KUKA KRL program: f1_Kuka_APT224T02S24.SRC

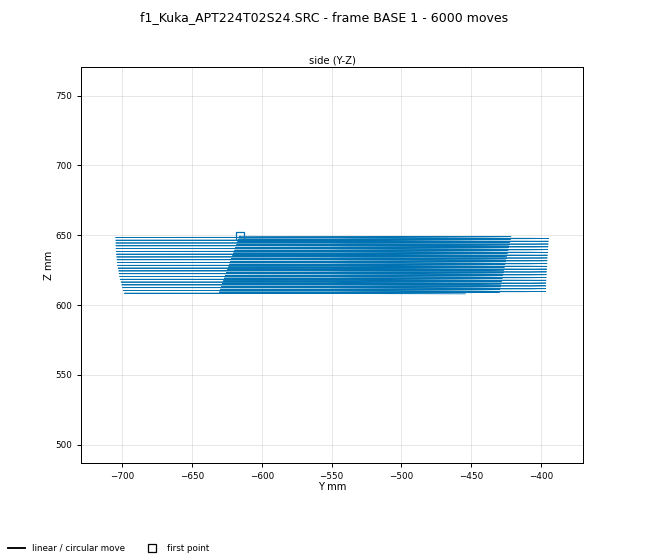
[picture p0: tool path of f1_Kuka_APT224T02S24.SRC in frame BASE 1, 6000 of 6001 moves have a stored position in this frame; points joined in program order, loops and branches not executed]
&ACCESS RVP
&REL 2
&PARAM TEMPLATE = C:\KRC\Roboter\Template\vorgabe
&PARAM EDITMASK = *
DEF f1_Kuka_APT224T02S24()


;FOLD INI;%{PE}%V3.2.0,%MKUKATPBASIS,%CINIT,%VCOMMON,%P
  ;FOLD BAS INI;%{E}%V3.2.0,%MKUKATPBASIS,%CINIT,%VINIT,%P
    GLOBAL INTERRUPT DECL 3 WHEN $STOPMESS==TRUE DO IR_STOPM ( )
    INTERRUPT ON 3
    BAS (#INITMOV,0 )
  ;ENDFOLD (BAS INI)
  ;FOLD USER INI;%{E}%V3.2.0,%MKUKATPUSER,%CINIT,%VINIT,%P
    ;Make your modifications here
  ;ENDFOLD (USER INI)
;ENDFOLD (INI)


;*** Make Null PTP Move
  PTP $pos_act

;*** Auto Load The Correct TOOL Data
  $tool=tool_data[2]

;*** Auto Load The Correct BASE Data
  $base=base_data[1]

  $ADVANCE = 5

;*** Restate Last Velocity
MMPM(30000.0)
SetRPM(8000)
LIN {X -0.107,Y -615.683,Z 649.293,A 0.000,B 0.000,C 90.000,E1 88.740} C_DIS
LIN {X -0.106,Y -616.052,Z 649.287,A 0.000,B 0.000,C 90.000,E1 87.707} C_DIS
LIN {X -0.093,Y -616.149,Z 649.281,A 0.000,B 0.000,C 90.000,E1 86.674} C_DIS
LIN {X 0.216,Y -615.988,Z 649.274,A 0.000,B 0.000,C 90.000,E1 85.355} C_DIS
LIN {X -0.079,Y -615.700,Z 649.270,A 0.000,B 0.000,C 90.000,E1 84.609} C_DIS
LIN {X -0.285,Y -615.137,Z 649.263,A 0.000,B 0.000,C 90.000,E1 83.337} C_DIS
LIN {X 0.118,Y -614.273,Z 649.256,A 0.000,B 0.000,C 90.000,E1 82.008} C_DIS
LIN {X 0.144,Y -613.216,Z 649.250,A 0.000,B 0.000,C 90.000,E1 80.971} C_DIS
LIN {X -0.008,Y -611.675,Z 649.243,A 0.000,B 0.000,C 90.000,E1 79.690} C_DIS
LIN {X -0.187,Y -609.834,Z 649.236,A 0.000,B 0.000,C 90.000,E1 78.409} C_DIS
LIN {X -0.275,Y -607.853,Z 649.228,A 0.000,B 0.000,C 90.000,E1 77.117} C_DIS
LIN {X 0.076,Y -605.171,Z 649.220,A 0.000,B 0.000,C 90.000,E1 75.519} C_DIS
LIN {X 0.063,Y -602.718,Z 649.212,A 0.000,B 0.000,C 90.000,E1 74.212} C_DIS
LIN {X 0.000,Y -600.058,Z 649.205,A 0.000,B 0.000,C 90.000,E1 72.906} C_DIS
LIN {X 0.062,Y -597.213,Z 649.198,A 0.000,B 0.000,C 90.000,E1 71.583} C_DIS
LIN {X 0.116,Y -595.336,Z 649.193,A 0.000,B 0.000,C 90.000,E1 70.786} C_DIS
LIN {X -0.045,Y -593.298,Z 649.189,A 0.000,B 0.000,C 90.000,E1 70.007} C_DIS
LIN {X -0.139,Y -590.246,Z 649.183,A 0.000,B 0.000,C 90.000,E1 68.954} C_DIS
LIN {X -0.032,Y -588.640,Z 649.180,A 0.000,B 0.000,C 90.000,E1 68.411} C_DIS
LIN {X -0.186,Y -584.996,Z 649.174,A 0.000,B 0.000,C 90.000,E1 67.358} C_DIS
LIN {X -0.157,Y -580.935,Z 649.168,A 0.000,B 0.000,C 90.000,E1 66.282} C_DIS
LIN {X -0.274,Y -577.678,Z 649.164,A 0.000,B 0.000,C 90.000,E1 65.485} C_DIS
LIN {X -0.191,Y -574.318,Z 649.159,A 0.000,B 0.000,C 90.000,E1 64.665} C_DIS
LIN {X 0.103,Y -570.576,Z 649.155,A 0.000,B 0.000,C 90.000,E1 63.819} C_DIS
LIN {X 0.189,Y -567.295,Z 649.151,A 0.000,B 0.000,C 90.000,E1 63.127} C_DIS
LIN {X -0.261,Y -563.689,Z 649.147,A 0.000,B 0.000,C 90.000,E1 62.487} C_DIS
LIN {X 0.018,Y -559.681,Z 649.143,A 0.000,B 0.000,C 90.000,E1 61.769} C_DIS
LIN {X 0.259,Y -555.194,Z 649.139,A 0.000,B 0.000,C 90.000,E1 61.051} C_DIS
LIN {X -0.181,Y -551.142,Z 649.136,A 0.000,B 0.000,C 90.000,E1 60.539} C_DIS
LIN {X 0.098,Y -546.732,Z 649.133,A 0.000,B 0.000,C 90.000,E1 59.950} C_DIS
LIN {X -0.119,Y -541.775,Z 649.130,A 0.000,B 0.000,C 90.000,E1 59.410} C_DIS
LIN {X -0.156,Y -537.571,Z 649.128,A 0.000,B 0.000,C 90.000,E1 58.997} C_DIS
LIN {X 0.112,Y -531.705,Z 649.125,A 0.000,B 0.000,C 90.000,E1 58.456} C_DIS
LIN {X 0.085,Y -525.967,Z 649.122,A 0.000,B 0.000,C 90.000,E1 57.995} C_DIS
LIN {X 0.245,Y -521.337,Z 649.121,A 0.000,B 0.000,C 90.000,E1 57.661} C_DIS
LIN {X -0.035,Y -515.202,Z 649.118,A 0.000,B 0.000,C 90.000,E1 57.296} C_DIS
LIN {X -0.193,Y -508.231,Z 649.116,A 0.000,B 0.000,C 90.000,E1 56.914} C_DIS
LIN {X 0.225,Y -501.476,Z 649.114,A 0.000,B 0.000,C 90.000,E1 56.501} C_DIS
LIN {X -0.128,Y -484.846,Z 649.109,A 0.000,B 0.000,C 90.000,E1 55.674} C_DIS
LIN {X -0.111,Y -464.619,Z 649.103,A 0.000,B 0.000,C 90.000,E1 54.609} C_DIS
LIN {X 0.001,Y -443.164,Z 649.097,A 0.000,B 0.000,C 90.000,E1 53.417} C_DIS
LIN {X -0.090,Y -435.744,Z 649.094,A 0.000,B 0.000,C 90.000,E1 53.004} C_DIS
LIN {X 0.128,Y -435.681,Z 649.094,A 0.000,B 0.000,C 90.000,E1 52.970} C_DIS
LIN {X -0.013,Y -431.775,Z 649.083,A 0.000,B 0.000,C 90.000,E1 50.964} C_DIS
LIN {X 0.166,Y -430.198,Z 649.079,A 0.000,B 0.000,C 90.000,E1 50.275} C_DIS
LIN {X -0.142,Y -421.586,Z 649.058,A 0.000,B 0.000,C 90.000,E1 46.458} C_DIS
LIN {X -0.193,Y -421.525,Z 649.057,A 0.000,B 0.000,C 90.000,E1 46.296} C_DIS
LIN {X -0.119,Y -421.750,Z 649.048,A 0.000,B 0.000,C 90.000,E1 44.595} C_DIS
LIN {X -0.046,Y -421.951,Z 649.038,A 0.000,B 0.000,C 90.000,E1 42.894} C_DIS
LIN {X 0.082,Y -422.604,Z 649.023,A 0.000,B 0.000,C 90.000,E1 40.172} C_DIS
LIN {X -0.082,Y -423.806,Z 649.006,A 0.000,B 0.000,C 90.000,E1 37.156} C_DIS
LIN {X 0.166,Y -424.678,Z 648.997,A 0.000,B 0.000,C 90.000,E1 35.438} C_DIS
LIN {X -0.039,Y -425.347,Z 648.990,A 0.000,B 0.000,C 90.000,E1 34.119} C_DIS
LIN {X 0.106,Y -426.158,Z 648.980,A 0.000,B 0.000,C 90.000,E1 32.418} C_DIS
LIN {X 0.029,Y -427.258,Z 648.967,A 0.000,B 0.000,C 90.000,E1 30.079} C_DIS
LIN {X -0.008,Y -427.926,Z 648.960,A 0.000,B 0.000,C 90.000,E1 28.743} C_DIS
LIN {X -0.083,Y -428.992,Z 648.949,A 0.000,B 0.000,C 90.000,E1 26.744} C_DIS
LIN {X 0.066,Y -430.831,Z 648.932,A 0.000,B 0.000,C 90.000,E1 23.718} C_DIS
LIN {X 0.087,Y -432.393,Z 648.921,A 0.000,B 0.000,C 90.000,E1 21.716} C_DIS
LIN {X -0.054,Y -433.161,Z 648.915,A 0.000,B 0.000,C 90.000,E1 20.737} C_DIS
LIN {X 0.047,Y -434.093,Z 648.908,A 0.000,B 0.000,C 90.000,E1 19.396} C_DIS
LIN {X 0.137,Y -435.669,Z 648.893,A 0.000,B 0.000,C 90.000,E1 16.732} C_DIS
LIN {X -0.050,Y -436.994,Z 648.882,A 0.000,B 0.000,C 90.000,E1 14.773} C_DIS
LIN {X 0.115,Y -438.556,Z 648.871,A 0.000,B 0.000,C 90.000,E1 12.771} C_DIS
LIN {X -0.052,Y -440.572,Z 648.858,A 0.000,B 0.000,C 90.000,E1 10.489} C_DIS
LIN {X 0.025,Y -442.495,Z 648.847,A 0.000,B 0.000,C 90.000,E1 8.511} C_DIS
LIN {X 0.187,Y -444.996,Z 648.835,A 0.000,B 0.000,C 90.000,E1 6.201} C_DIS
LIN {X -0.078,Y -447.653,Z 648.822,A 0.000,B 0.000,C 90.000,E1 3.955} C_DIS
LIN {X -0.219,Y -449.744,Z 648.813,A 0.000,B 0.000,C 90.000,E1 2.350} C_DIS
LIN {X 0.000,Y -452.970,Z 648.800,A 0.000,B 0.000,C 90.000,E1 360.000} C_DIS
LIN {X -0.220,Y -457.336,Z 648.785,A 0.000,B 0.000,C 90.000,E1 357.249} C_DIS
LIN {X 0.046,Y -460.604,Z 648.774,A 0.000,B 0.000,C 90.000,E1 355.298} C_DIS
LIN {X 0.014,Y -463.997,Z 648.763,A 0.000,B 0.000,C 90.000,E1 353.394} C_DIS
LIN {X -0.200,Y -466.761,Z 648.755,A 0.000,B 0.000,C 90.000,E1 351.837} C_DIS
LIN {X -0.041,Y -469.029,Z 648.748,A 0.000,B 0.000,C 90.000,E1 350.557} C_DIS
LIN {X 0.182,Y -472.299,Z 648.737,A 0.000,B 0.000,C 90.000,E1 348.645} C_DIS
LIN {X 0.135,Y -476.180,Z 648.725,A 0.000,B 0.000,C 90.000,E1 346.464} C_DIS
LIN {X -0.113,Y -479.645,Z 648.715,A 0.000,B 0.000,C 90.000,E1 344.629} C_DIS
LIN {X -0.159,Y -483.757,Z 648.703,A 0.000,B 0.000,C 90.000,E1 342.472} C_DIS
LIN {X 0.014,Y -486.192,Z 648.696,A 0.000,B 0.000,C 90.000,E1 341.221} C_DIS
LIN {X -0.016,Y -490.429,Z 648.684,A 0.000,B 0.000,C 90.000,E1 339.082} C_DIS
LIN {X 0.161,Y -493.332,Z 648.675,A 0.000,B 0.000,C 90.000,E1 337.539} C_DIS
LIN {X -0.115,Y -495.497,Z 648.669,A 0.000,B 0.000,C 90.000,E1 336.357} C_DIS
LIN {X 0.032,Y -497.016,Z 648.664,A 0.000,B 0.000,C 90.000,E1 335.433} C_DIS
LIN {X -0.110,Y -499.995,Z 648.654,A 0.000,B 0.000,C 90.000,E1 333.640} C_DIS
LIN {X -0.266,Y -504.032,Z 648.640,A 0.000,B 0.000,C 90.000,E1 331.257} C_DIS
LIN {X -0.088,Y -506.996,Z 648.632,A 0.000,B 0.000,C 90.000,E1 329.744} C_DIS
LIN {X 0.118,Y -508.525,Z 648.629,A 0.000,B 0.000,C 90.000,E1 329.125} C_DIS
LIN {X -0.253,Y -509.466,Z 648.627,A 0.000,B 0.000,C 90.000,E1 328.869} C_DIS
LIN {X 0.077,Y -510.694,Z 648.625,A 0.000,B 0.000,C 90.000,E1 328.535} C_DIS
LIN {X -0.021,Y -511.789,Z 648.624,A 0.000,B 0.000,C 90.000,E1 328.250} C_DIS
LIN {X 0.048,Y -513.255,Z 648.622,A 0.000,B 0.000,C 90.000,E1 327.946} C_DIS
LIN {X 0.057,Y -516.255,Z 648.620,A 0.000,B 0.000,C 90.000,E1 327.502} C_DIS
LIN {X 0.011,Y -521.889,Z 648.616,A 0.000,B 0.000,C 90.000,E1 326.914} C_DIS
LIN {X -0.112,Y -525.881,Z 648.614,A 0.000,B 0.000,C 90.000,E1 326.580} C_DIS
LIN {X 0.283,Y -537.745,Z 648.609,A 0.000,B 0.000,C 90.000,E1 325.595} C_DIS
LIN {X 0.056,Y -549.203,Z 648.604,A 0.000,B 0.000,C 90.000,E1 324.689} C_DIS
LIN {X -0.222,Y -556.292,Z 648.601,A 0.000,B 0.000,C 90.000,E1 324.116} C_DIS
LIN {X -0.114,Y -563.209,Z 648.597,A 0.000,B 0.000,C 90.000,E1 323.497} C_DIS
LIN {X 0.017,Y -571.227,Z 648.593,A 0.000,B 0.000,C 90.000,E1 322.763} C_DIS
LIN {X 0.042,Y -577.842,Z 648.590,A 0.000,B 0.000,C 90.000,E1 322.145} C_DIS
LIN {X 0.149,Y -589.774,Z 648.583,A 0.000,B 0.000,C 90.000,E1 321.009} C_DIS
LIN {X 0.118,Y -598.681,Z 648.579,A 0.000,B 0.000,C 90.000,E1 320.150} C_DIS
LIN {X 0.160,Y -603.373,Z 648.576,A 0.000,B 0.000,C 90.000,E1 319.666} C_DIS
LIN {X -0.061,Y -607.139,Z 648.574,A 0.000,B 0.000,C 90.000,E1 319.299} C_DIS
LIN {X 0.343,Y -611.567,Z 648.571,A 0.000,B 0.000,C 90.000,E1 318.771} C_DIS
LIN {X 0.191,Y -614.856,Z 648.569,A 0.000,B 0.000,C 90.000,E1 318.405} C_DIS
LIN {X -0.339,Y -622.061,Z 648.564,A 0.000,B 0.000,C 90.000,E1 317.553} C_DIS
LIN {X 0.120,Y -627.754,Z 648.560,A 0.000,B 0.000,C 90.000,E1 316.743} C_DIS
LIN {X 0.330,Y -631.363,Z 648.557,A 0.000,B 0.000,C 90.000,E1 316.215} C_DIS
LIN {X 0.001,Y -636.638,Z 648.553,A 0.000,B 0.000,C 90.000,E1 315.486} C_DIS
LIN {X -0.361,Y -643.266,Z 648.547,A 0.000,B 0.000,C 90.000,E1 314.514} C_DIS
LIN {X 0.045,Y -648.774,Z 648.542,A 0.000,B 0.000,C 90.000,E1 313.623} C_DIS
LIN {X -0.125,Y -653.467,Z 648.538,A 0.000,B 0.000,C 90.000,E1 312.894} C_DIS
LIN {X -0.212,Y -657.818,Z 648.534,A 0.000,B 0.000,C 90.000,E1 312.162} C_DIS
LIN {X -0.285,Y -662.565,Z 648.529,A 0.000,B 0.000,C 90.000,E1 311.310} C_DIS
LIN {X -0.311,Y -667.018,Z 648.525,A 0.000,B 0.000,C 90.000,E1 310.458} C_DIS
LIN {X -0.255,Y -670.469,Z 648.521,A 0.000,B 0.000,C 90.000,E1 309.725} C_DIS
LIN {X 0.262,Y -672.625,Z 648.518,A 0.000,B 0.000,C 90.000,E1 309.197} C_DIS
LIN {X 0.377,Y -675.571,Z 648.514,A 0.000,B 0.000,C 90.000,E1 308.463} C_DIS
LIN {X -0.025,Y -677.423,Z 648.511,A 0.000,B 0.000,C 90.000,E1 308.016} C_DIS
LIN {X -0.264,Y -680.708,Z 648.506,A 0.000,B 0.000,C 90.000,E1 307.076} C_DIS
LIN {X 0.086,Y -683.783,Z 648.501,A 0.000,B 0.000,C 90.000,E1 306.091} C_DIS
LIN {X -0.263,Y -687.978,Z 648.493,A 0.000,B 0.000,C 90.000,E1 304.692} C_DIS
LIN {X -0.179,Y -691.158,Z 648.486,A 0.000,B 0.000,C 90.000,E1 303.499} C_DIS
LIN {X 0.154,Y -694.085,Z 648.479,A 0.000,B 0.000,C 90.000,E1 302.291} C_DIS
LIN {X -0.053,Y -696.738,Z 648.473,A 0.000,B 0.000,C 90.000,E1 301.131} C_DIS
LIN {X 0.019,Y -699.078,Z 648.466,A 0.000,B 0.000,C 90.000,E1 299.951} C_DIS
LIN {X 0.138,Y -701.185,Z 648.460,A 0.000,B 0.000,C 90.000,E1 298.771} C_DIS
LIN {X 0.008,Y -702.635,Z 648.455,A 0.000,B 0.000,C 90.000,E1 297.847} C_DIS
LIN {X -0.118,Y -703.897,Z 648.450,A 0.000,B 0.000,C 90.000,E1 296.924} C_DIS
LIN {X -0.209,Y -704.731,Z 648.446,A 0.000,B 0.000,C 90.000,E1 296.232} C_DIS
LIN {X 0.366,Y -704.865,Z 648.443,A 0.000,B 0.000,C 90.000,E1 295.720} C_DIS
LIN {X -0.286,Y -704.814,Z 648.442,A 0.000,B 0.000,C 90.000,E1 295.540} C_DIS
LIN {X 0.290,Y -704.038,Z 648.439,A 0.000,B 0.000,C 90.000,E1 295.027} C_DIS
LIN {X -0.063,Y -703.354,Z 648.438,A 0.000,B 0.000,C 90.000,E1 294.823} C_DIS
LIN {X 0.206,Y -700.408,Z 648.435,A 0.000,B 0.000,C 90.000,E1 294.335} C_DIS
LIN {X 0.342,Y -699.590,Z 648.435,A 0.000,B 0.000,C 90.000,E1 294.207} C_DIS
LIN {X -0.160,Y -698.417,Z 648.434,A 0.000,B 0.000,C 90.000,E1 294.131} C_DIS
LIN {X -0.024,Y -696.601,Z 648.433,A 0.000,B 0.000,C 90.000,E1 294.003} C_DIS
LIN {X -0.402,Y -690.632,Z 648.432,A 0.000,B 0.000,C 90.000,E1 293.770} C_DIS
LIN {X 0.296,Y -688.546,Z 648.432,A 0.000,B 0.000,C 90.000,E1 293.643} C_DIS
LIN {X -0.197,Y -683.792,Z 648.431,A 0.000,B 0.000,C 90.000,E1 293.567} C_DIS
LIN {X -0.125,Y -681.698,Z 648.431,A 0.000,B 0.000,C 90.000,E1 293.515} C_DIS
LIN {X -0.168,Y -675.378,Z 648.430,A 0.000,B 0.000,C 90.000,E1 293.439} C_DIS
LIN {X -0.316,Y -664.050,Z 648.430,A 0.000,B 0.000,C 90.000,E1 293.334} C_DIS
LIN {X 0.192,Y -653.634,Z 648.429,A 0.000,B 0.000,C 90.000,E1 293.153} C_DIS
LIN {X -0.065,Y -640.843,Z 648.427,A 0.000,B 0.000,C 90.000,E1 292.950} C_DIS
LIN {X 0.153,Y -630.607,Z 648.426,A 0.000,B 0.000,C 90.000,E1 292.717} C_DIS
LIN {X 0.120,Y -617.705,Z 648.424,A 0.000,B 0.000,C 90.000,E1 292.386} C_DIS
LIN {X -0.192,Y -590.387,Z 648.420,A 0.000,B 0.000,C 90.000,E1 291.589} C_DIS
LIN {X 0.092,Y -578.237,Z 648.418,A 0.000,B 0.000,C 90.000,E1 291.173} C_DIS
LIN {X -0.153,Y -564.169,Z 648.415,A 0.000,B 0.000,C 90.000,E1 290.791} C_DIS
LIN {X -0.215,Y -560.765,Z 648.415,A 0.000,B 0.000,C 90.000,E1 290.663} C_DIS
LIN {X 0.178,Y -559.398,Z 648.414,A 0.000,B 0.000,C 90.000,E1 290.556} C_DIS
LIN {X -0.320,Y -556.686,Z 648.413,A 0.000,B 0.000,C 90.000,E1 290.429} C_DIS
LIN {X 0.158,Y -556.628,Z 648.413,A 0.000,B 0.000,C 90.000,E1 290.375} C_DIS
LIN {X -0.272,Y -555.838,Z 648.412,A 0.000,B 0.000,C 90.000,E1 290.248} C_DIS
LIN {X -0.096,Y -555.284,Z 648.410,A 0.000,B 0.000,C 90.000,E1 289.812} C_DIS
LIN {X 0.141,Y -555.127,Z 648.401,A 0.000,B 0.000,C 90.000,E1 288.127} C_DIS
LIN {X -0.127,Y -554.919,Z 648.395,A 0.000,B 0.000,C 90.000,E1 287.040} C_DIS
LIN {X 0.244,Y -554.482,Z 648.387,A 0.000,B 0.000,C 90.000,E1 285.607} C_DIS
LIN {X -0.075,Y -553.872,Z 648.379,A 0.000,B 0.000,C 90.000,E1 284.245} C_DIS
LIN {X 0.132,Y -553.079,Z 648.371,A 0.000,B 0.000,C 90.000,E1 282.827} C_DIS
LIN {X -0.221,Y -552.260,Z 648.362,A 0.000,B 0.000,C 90.000,E1 281.186} C_DIS
LIN {X -0.036,Y -551.416,Z 648.351,A 0.000,B 0.000,C 90.000,E1 279.208} C_DIS
LIN {X -0.103,Y -550.974,Z 648.343,A 0.000,B 0.000,C 90.000,E1 277.814} C_DIS
LIN {X -0.070,Y -550.369,Z 648.331,A 0.000,B 0.000,C 90.000,E1 275.568} C_DIS
LIN {X -0.196,Y -549.990,Z 648.322,A 0.000,B 0.000,C 90.000,E1 273.898} C_DIS
LIN {X 0.039,Y -549.768,Z 648.315,A 0.000,B 0.000,C 90.000,E1 272.751} C_DIS
LIN {X -0.227,Y -549.355,Z 648.308,A 0.000,B 0.000,C 90.000,E1 271.375} C_DIS
LIN {X 0.089,Y -548.641,Z 648.298,A 0.000,B 0.000,C 90.000,E1 269.656} C_DIS
LIN {X -0.099,Y -547.616,Z 648.287,A 0.000,B 0.000,C 90.000,E1 267.707} C_DIS
LIN {X 0.146,Y -546.923,Z 648.279,A 0.000,B 0.000,C 90.000,E1 266.274} C_DIS
LIN {X -0.168,Y -546.194,Z 648.273,A 0.000,B 0.000,C 90.000,E1 265.179} C_DIS
LIN {X 0.105,Y -544.936,Z 648.264,A 0.000,B 0.000,C 90.000,E1 263.457} C_DIS
LIN {X -0.170,Y -543.835,Z 648.258,A 0.000,B 0.000,C 90.000,E1 262.356} C_DIS
LIN {X 0.168,Y -542.255,Z 648.250,A 0.000,B 0.000,C 90.000,E1 260.905} C_DIS
LIN {X 0.249,Y -539.825,Z 648.235,A 0.000,B 0.000,C 90.000,E1 258.342} C_DIS
LIN {X -0.247,Y -537.852,Z 648.223,A 0.000,B 0.000,C 90.000,E1 256.117} C_DIS
LIN {X -0.196,Y -536.646,Z 648.215,A 0.000,B 0.000,C 90.000,E1 254.685} C_DIS
LIN {X -0.112,Y -535.006,Z 648.205,A 0.000,B 0.000,C 90.000,E1 252.960} C_DIS
LIN {X 0.278,Y -533.146,Z 648.194,A 0.000,B 0.000,C 90.000,E1 250.913} C_DIS
LIN {X 0.190,Y -532.156,Z 648.189,A 0.000,B 0.000,C 90.000,E1 250.061} C_DIS
LIN {X -0.211,Y -530.582,Z 648.183,A 0.000,B 0.000,C 90.000,E1 248.954} C_DIS
LIN {X 0.041,Y -528.498,Z 648.175,A 0.000,B 0.000,C 90.000,E1 247.486} C_DIS
LIN {X -0.212,Y -526.670,Z 648.169,A 0.000,B 0.000,C 90.000,E1 246.357} C_DIS
LIN {X -0.102,Y -524.052,Z 648.161,A 0.000,B 0.000,C 90.000,E1 244.897} C_DIS
LIN {X 0.051,Y -521.740,Z 648.154,A 0.000,B 0.000,C 90.000,E1 243.717} C_DIS
LIN {X -0.166,Y -518.703,Z 648.146,A 0.000,B 0.000,C 90.000,E1 242.281} C_DIS
LIN {X 0.026,Y -515.645,Z 648.138,A 0.000,B 0.000,C 90.000,E1 240.795} C_DIS
LIN {X -0.042,Y -512.300,Z 648.130,A 0.000,B 0.000,C 90.000,E1 239.331} C_DIS
LIN {X -0.170,Y -508.899,Z 648.121,A 0.000,B 0.000,C 90.000,E1 237.867} C_DIS
LIN {X -0.204,Y -504.729,Z 648.112,A 0.000,B 0.000,C 90.000,E1 236.087} C_DIS
LIN {X 0.066,Y -500.858,Z 648.103,A 0.000,B 0.000,C 90.000,E1 234.562} C_DIS
LIN {X 0.149,Y -496.971,Z 648.095,A 0.000,B 0.000,C 90.000,E1 233.050} C_DIS
LIN {X 0.028,Y -490.996,Z 648.081,A 0.000,B 0.000,C 90.000,E1 230.642} C_DIS
LIN {X -0.161,Y -485.917,Z 648.070,A 0.000,B 0.000,C 90.000,E1 228.528} C_DIS
LIN {X -0.166,Y -480.801,Z 648.058,A 0.000,B 0.000,C 90.000,E1 226.377} C_DIS
LIN {X -0.110,Y -476.363,Z 648.047,A 0.000,B 0.000,C 90.000,E1 224.514} C_DIS
LIN {X -0.045,Y -471.265,Z 648.035,A 0.000,B 0.000,C 90.000,E1 222.324} C_DIS
LIN {X 0.231,Y -466.428,Z 648.023,A 0.000,B 0.000,C 90.000,E1 220.092} C_DIS
LIN {X 0.128,Y -461.737,Z 648.011,A 0.000,B 0.000,C 90.000,E1 217.890} C_DIS
LIN {X -0.011,Y -456.628,Z 647.996,A 0.000,B 0.000,C 90.000,E1 215.358} C_DIS
LIN {X -0.254,Y -453.661,Z 647.988,A 0.000,B 0.000,C 90.000,E1 213.785} C_DIS
LIN {X 0.249,Y -449.539,Z 647.975,A 0.000,B 0.000,C 90.000,E1 211.465} C_DIS
LIN {X -0.048,Y -447.227,Z 647.968,A 0.000,B 0.000,C 90.000,E1 210.207} C_DIS
LIN {X 0.012,Y -444.957,Z 647.961,A 0.000,B 0.000,C 90.000,E1 208.899} C_DIS
LIN {X -0.067,Y -441.381,Z 647.950,A 0.000,B 0.000,C 90.000,E1 206.950} C_DIS
LIN {X 0.149,Y -437.814,Z 647.939,A 0.000,B 0.000,C 90.000,E1 204.951} C_DIS
LIN {X -0.105,Y -434.164,Z 647.928,A 0.000,B 0.000,C 90.000,E1 203.003} C_DIS
LIN {X -0.030,Y -431.226,Z 647.919,A 0.000,B 0.000,C 90.000,E1 201.334} C_DIS
LIN {X 0.235,Y -428.339,Z 647.909,A 0.000,B 0.000,C 90.000,E1 199.631} C_DIS
LIN {X 0.109,Y -426.094,Z 647.902,A 0.000,B 0.000,C 90.000,E1 198.308} C_DIS
LIN {X -0.077,Y -422.726,Z 647.891,A 0.000,B 0.000,C 90.000,E1 196.315} C_DIS
LIN {X 0.168,Y -420.067,Z 647.881,A 0.000,B 0.000,C 90.000,E1 194.592} C_DIS
LIN {X -0.154,Y -417.378,Z 647.872,A 0.000,B 0.000,C 90.000,E1 192.939} C_DIS
LIN {X -0.119,Y -413.706,Z 647.859,A 0.000,B 0.000,C 90.000,E1 190.546} C_DIS
LIN {X 0.120,Y -410.693,Z 647.847,A 0.000,B 0.000,C 90.000,E1 188.454} C_DIS
LIN {X -0.205,Y -408.163,Z 647.838,A 0.000,B 0.000,C 90.000,E1 186.777} C_DIS
LIN {X 0.187,Y -405.323,Z 647.826,A 0.000,B 0.000,C 90.000,E1 184.645} C_DIS
LIN {X -0.058,Y -401.625,Z 647.809,A 0.000,B 0.000,C 90.000,E1 181.547} C_DIS
LIN {X -0.099,Y -398.423,Z 647.789,A 0.000,B 0.000,C 90.000,E1 178.051} C_DIS
LIN {X 0.130,Y -396.099,Z 647.768,A 0.000,B 0.000,C 90.000,E1 174.147} C_DIS
LIN {X -0.107,Y -395.294,Z 647.756,A 0.000,B 0.000,C 90.000,E1 172.064} C_DIS
LIN {X 0.026,Y -394.834,Z 647.744,A 0.000,B 0.000,C 90.000,E1 169.926} C_DIS
LIN {X -0.109,Y -394.571,Z 647.728,A 0.000,B 0.000,C 90.000,E1 167.117} C_DIS
LIN {X -0.079,Y -394.593,Z 647.717,A 0.000,B 0.000,C 90.000,E1 164.991} C_DIS
LIN {X 0.051,Y -394.832,Z 647.705,A 0.000,B 0.000,C 90.000,E1 162.851} C_DIS
LIN {X 0.043,Y -395.183,Z 647.693,A 0.000,B 0.000,C 90.000,E1 160.732} C_DIS
LIN {X 0.183,Y -395.589,Z 647.681,A 0.000,B 0.000,C 90.000,E1 158.592} C_DIS
LIN {X 0.109,Y -396.088,Z 647.669,A 0.000,B 0.000,C 90.000,E1 156.485} C_DIS
LIN {X 0.060,Y -396.697,Z 647.656,A 0.000,B 0.000,C 90.000,E1 154.024} C_DIS
LIN {X 0.153,Y -397.211,Z 647.644,A 0.000,B 0.000,C 90.000,E1 151.897} C_DIS
LIN {X -0.024,Y -397.822,Z 647.630,A 0.000,B 0.000,C 90.000,E1 149.459} C_DIS
LIN {X -0.080,Y -398.335,Z 647.621,A 0.000,B 0.000,C 90.000,E1 147.709} C_DIS
LIN {X 0.087,Y -398.967,Z 647.611,A 0.000,B 0.000,C 90.000,E1 145.928} C_DIS
LIN {X -0.083,Y -399.969,Z 647.597,A 0.000,B 0.000,C 90.000,E1 143.497} C_DIS
LIN {X -0.069,Y -400.793,Z 647.587,A 0.000,B 0.000,C 90.000,E1 141.743} C_DIS
LIN {X 0.083,Y -401.734,Z 647.576,A 0.000,B 0.000,C 90.000,E1 139.622} C_DIS
LIN {X 0.077,Y -402.545,Z 647.566,A 0.000,B 0.000,C 90.000,E1 137.877} C_DIS
LIN {X -0.110,Y -403.508,Z 647.554,A 0.000,B 0.000,C 90.000,E1 135.810} C_DIS
LIN {X 0.012,Y -404.522,Z 647.543,A 0.000,B 0.000,C 90.000,E1 133.704} C_DIS
LIN {X 0.035,Y -405.539,Z 647.533,A 0.000,B 0.000,C 90.000,E1 131.962} C_DIS
LIN {X 0.000,Y -406.174,Z 647.529,A 0.000,B 0.000,C 90.000,E1 131.272} C_DIS
LIN {X -0.154,Y -407.518,Z 647.524,A 0.000,B 0.000,C 90.000,E1 130.253} C_DIS
LIN {X -0.008,Y -408.461,Z 647.522,A 0.000,B 0.000,C 90.000,E1 129.886} C_DIS
LIN {X 0.103,Y -409.409,Z 647.519,A 0.000,B 0.000,C 90.000,E1 129.439} C_DIS
LIN {X 0.178,Y -411.840,Z 647.516,A 0.000,B 0.000,C 90.000,E1 128.910} C_DIS
LIN {X -0.196,Y -415.297,Z 647.514,A 0.000,B 0.000,C 90.000,E1 128.543} C_DIS
LIN {X -0.055,Y -419.154,Z 647.512,A 0.000,B 0.000,C 90.000,E1 128.177} C_DIS
LIN {X -0.173,Y -425.267,Z 647.510,A 0.000,B 0.000,C 90.000,E1 127.729} C_DIS
LIN {X 0.016,Y -448.346,Z 647.501,A 0.000,B 0.000,C 90.000,E1 126.171} C_DIS
LIN {X 0.021,Y -458.043,Z 647.497,A 0.000,B 0.000,C 90.000,E1 125.518} C_DIS
LIN {X -0.031,Y -469.125,Z 647.493,A 0.000,B 0.000,C 90.000,E1 124.739} C_DIS
LIN {X 0.026,Y -475.373,Z 647.490,A 0.000,B 0.000,C 90.000,E1 124.278} C_DIS
LIN {X -0.104,Y -483.063,Z 647.487,A 0.000,B 0.000,C 90.000,E1 123.706} C_DIS
LIN {X 0.067,Y -490.668,Z 647.484,A 0.000,B 0.000,C 90.000,E1 123.086} C_DIS
LIN {X -0.184,Y -496.543,Z 647.481,A 0.000,B 0.000,C 90.000,E1 122.625} C_DIS
LIN {X -0.098,Y -508.118,Z 647.476,A 0.000,B 0.000,C 90.000,E1 121.592} C_DIS
LIN {X 0.200,Y -516.460,Z 647.471,A 0.000,B 0.000,C 90.000,E1 120.797} C_DIS
LIN {X 0.127,Y -520.580,Z 647.469,A 0.000,B 0.000,C 90.000,E1 120.413} C_DIS
LIN {X 0.014,Y -528.558,Z 647.465,A 0.000,B 0.000,C 90.000,E1 119.617} C_DIS
LIN {X -0.153,Y -533.705,Z 647.461,A 0.000,B 0.000,C 90.000,E1 119.077} C_DIS
LIN {X 0.305,Y -539.291,Z 647.458,A 0.000,B 0.000,C 90.000,E1 118.359} C_DIS
LIN {X 0.122,Y -543.436,Z 647.455,A 0.000,B 0.000,C 90.000,E1 117.847} C_DIS
LIN {X -0.143,Y -547.345,Z 647.452,A 0.000,B 0.000,C 90.000,E1 117.308} C_DIS
LIN {X -0.051,Y -551.442,Z 647.448,A 0.000,B 0.000,C 90.000,E1 116.616} C_DIS
LIN {X 0.002,Y -555.950,Z 647.443,A 0.000,B 0.000,C 90.000,E1 115.771} C_DIS
LIN {X -0.141,Y -559.903,Z 647.439,A 0.000,B 0.000,C 90.000,E1 114.951} C_DIS
LIN {X -0.143,Y -562.943,Z 647.435,A 0.000,B 0.000,C 90.000,E1 114.259} C_DIS
LIN {X 0.106,Y -567.384,Z 647.429,A 0.000,B 0.000,C 90.000,E1 113.131} C_DIS
LIN {X -0.146,Y -570.506,Z 647.424,A 0.000,B 0.000,C 90.000,E1 112.333} C_DIS
LIN {X 0.171,Y -573.255,Z 647.419,A 0.000,B 0.000,C 90.000,E1 111.482} C_DIS
LIN {X 0.192,Y -575.721,Z 647.415,A 0.000,B 0.000,C 90.000,E1 110.663} C_DIS
LIN {X -0.169,Y -578.029,Z 647.410,A 0.000,B 0.000,C 90.000,E1 109.885} C_DIS
LIN {X 0.046,Y -579.483,Z 647.407,A 0.000,B 0.000,C 90.000,E1 109.322} C_DIS
LIN {X -0.228,Y -582.628,Z 647.400,A 0.000,B 0.000,C 90.000,E1 108.000} C_DIS
LIN {X -0.212,Y -586.087,Z 647.391,A 0.000,B 0.000,C 90.000,E1 106.386} C_DIS
LIN {X 0.132,Y -590.321,Z 647.381,A 0.000,B 0.000,C 90.000,E1 104.481} C_DIS
LIN {X 0.149,Y -593.963,Z 647.372,A 0.000,B 0.000,C 90.000,E1 102.883} C_DIS
LIN {X 0.109,Y -596.335,Z 647.366,A 0.000,B 0.000,C 90.000,E1 101.827} C_DIS
LIN {X 0.290,Y -600.355,Z 647.356,A 0.000,B 0.000,C 90.000,E1 99.962} C_DIS
LIN {X -0.062,Y -603.157,Z 647.348,A 0.000,B 0.000,C 90.000,E1 98.681} C_DIS
LIN {X -0.181,Y -605.260,Z 647.342,A 0.000,B 0.000,C 90.000,E1 97.644} C_DIS
LIN {X -0.263,Y -607.174,Z 647.337,A 0.000,B 0.000,C 90.000,E1 96.606} C_DIS
LIN {X 0.003,Y -609.361,Z 647.329,A 0.000,B 0.000,C 90.000,E1 95.277} C_DIS
LIN {X 0.242,Y -611.349,Z 647.322,A 0.000,B 0.000,C 90.000,E1 93.955} C_DIS
LIN {X 0.187,Y -612.797,Z 647.316,A 0.000,B 0.000,C 90.000,E1 92.922} C_DIS
LIN {X 0.129,Y -614.022,Z 647.311,A 0.000,B 0.000,C 90.000,E1 91.892} C_DIS
LIN {X -0.190,Y -614.808,Z 647.306,A 0.000,B 0.000,C 90.000,E1 91.146} C_DIS
LIN {X 0.089,Y -615.815,Z 647.299,A 0.000,B 0.000,C 90.000,E1 89.828} C_DIS
LIN {X -0.228,Y -616.260,Z 647.295,A 0.000,B 0.000,C 90.000,E1 89.083} C_DIS
LIN {X 0.089,Y -616.764,Z 647.288,A 0.000,B 0.000,C 90.000,E1 87.764} C_DIS
LIN {X 0.111,Y -616.827,Z 647.282,A 0.000,B 0.000,C 90.000,E1 86.731} C_DIS
LIN {X -0.181,Y -616.696,Z 647.275,A 0.000,B 0.000,C 90.000,E1 85.469} C_DIS
LIN {X 0.147,Y -616.421,Z 647.271,A 0.000,B 0.000,C 90.000,E1 84.666} C_DIS
LIN {X -0.047,Y -615.798,Z 647.263,A 0.000,B 0.000,C 90.000,E1 83.394} C_DIS
LIN {X -0.324,Y -614.941,Z 647.256,A 0.000,B 0.000,C 90.000,E1 82.129} C_DIS
LIN {X -0.200,Y -613.884,Z 647.250,A 0.000,B 0.000,C 90.000,E1 81.084} C_DIS
LIN {X 0.267,Y -612.315,Z 647.243,A 0.000,B 0.000,C 90.000,E1 79.746} C_DIS
LIN {X 0.100,Y -610.454,Z 647.236,A 0.000,B 0.000,C 90.000,E1 78.465} C_DIS
LIN {X 0.025,Y -608.448,Z 647.229,A 0.000,B 0.000,C 90.000,E1 77.173} C_DIS
LIN {X -0.085,Y -606.179,Z 647.222,A 0.000,B 0.000,C 90.000,E1 75.880} C_DIS
LIN {X 0.182,Y -604.260,Z 647.216,A 0.000,B 0.000,C 90.000,E1 74.810} C_DIS
LIN {X -0.155,Y -602.179,Z 647.210,A 0.000,B 0.000,C 90.000,E1 73.795} C_DIS
LIN {X -0.230,Y -599.408,Z 647.203,A 0.000,B 0.000,C 90.000,E1 72.489} C_DIS
LIN {X 0.115,Y -597.073,Z 647.197,A 0.000,B 0.000,C 90.000,E1 71.402} C_DIS
LIN {X -0.137,Y -594.389,Z 647.191,A 0.000,B 0.000,C 90.000,E1 70.369} C_DIS
LIN {X 0.338,Y -591.421,Z 647.185,A 0.000,B 0.000,C 90.000,E1 69.263} C_DIS
LIN {X 0.338,Y -588.976,Z 647.181,A 0.000,B 0.000,C 90.000,E1 68.465} C_DIS
LIN {X 0.311,Y -586.224,Z 647.176,A 0.000,B 0.000,C 90.000,E1 67.667} C_DIS
LIN {X 0.121,Y -582.204,Z 647.170,A 0.000,B 0.000,C 90.000,E1 66.613} C_DIS
LIN {X 0.250,Y -578.977,Z 647.166,A 0.000,B 0.000,C 90.000,E1 65.793} C_DIS
LIN {X 0.197,Y -574.425,Z 647.160,A 0.000,B 0.000,C 90.000,E1 64.717} C_DIS
LIN {X 0.240,Y -570.643,Z 647.155,A 0.000,B 0.000,C 90.000,E1 63.896} C_DIS
LIN {X -0.270,Y -566.530,Z 647.151,A 0.000,B 0.000,C 90.000,E1 63.127} C_DIS
LIN {X 0.035,Y -562.765,Z 647.147,A 0.000,B 0.000,C 90.000,E1 62.410} C_DIS
LIN {X 0.142,Y -559.496,Z 647.144,A 0.000,B 0.000,C 90.000,E1 61.847} C_DIS
LIN {X -0.108,Y -554.936,Z 647.140,A 0.000,B 0.000,C 90.000,E1 61.179} C_DIS
LIN {X -0.120,Y -550.920,Z 647.137,A 0.000,B 0.000,C 90.000,E1 60.639} C_DIS
LIN {X -0.308,Y -545.531,Z 647.133,A 0.000,B 0.000,C 90.000,E1 59.999} C_DIS
LIN {X 0.104,Y -541.018,Z 647.130,A 0.000,B 0.000,C 90.000,E1 59.459} C_DIS
LIN {X -0.029,Y -536.896,Z 647.128,A 0.000,B 0.000,C 90.000,E1 59.076} C_DIS
LIN {X -0.163,Y -531.283,Z 647.126,A 0.000,B 0.000,C 90.000,E1 58.614} C_DIS
LIN {X -0.037,Y -525.229,Z 647.123,A 0.000,B 0.000,C 90.000,E1 58.122} C_DIS
LIN {X 0.149,Y -518.547,Z 647.120,A 0.000,B 0.000,C 90.000,E1 57.661} C_DIS
LIN {X 0.014,Y -513.657,Z 647.119,A 0.000,B 0.000,C 90.000,E1 57.375} C_DIS
LIN {X 0.032,Y -506.897,Z 647.117,A 0.000,B 0.000,C 90.000,E1 56.993} C_DIS
LIN {X 0.066,Y -500.070,Z 647.115,A 0.000,B 0.000,C 90.000,E1 56.628} C_DIS
LIN {X -0.261,Y -484.938,Z 647.110,A 0.000,B 0.000,C 90.000,E1 55.881} C_DIS
LIN {X 0.101,Y -463.040,Z 647.104,A 0.000,B 0.000,C 90.000,E1 54.689} C_DIS
LIN {X -0.159,Y -443.026,Z 647.098,A 0.000,B 0.000,C 90.000,E1 53.623} C_DIS
LIN {X 0.052,Y -436.235,Z 647.096,A 0.000,B 0.000,C 90.000,E1 53.210} C_DIS
LIN {X 0.008,Y -436.154,Z 647.096,A 0.000,B 0.000,C 90.000,E1 53.210} C_DIS
LIN {X 0.094,Y -431.511,Z 647.082,A 0.000,B 0.000,C 90.000,E1 50.803} C_DIS
LIN {X 0.053,Y -421.953,Z 647.059,A 0.000,B 0.000,C 90.000,E1 46.620} C_DIS
LIN {X 0.188,Y -422.233,Z 647.051,A 0.000,B 0.000,C 90.000,E1 45.081} C_DIS
LIN {X -0.221,Y -422.513,Z 647.037,A 0.000,B 0.000,C 90.000,E1 42.771} C_DIS
LIN {X -0.006,Y -423.118,Z 647.024,A 0.000,B 0.000,C 90.000,E1 40.378} C_DIS
LIN {X -0.158,Y -424.334,Z 647.008,A 0.000,B 0.000,C 90.000,E1 37.363} C_DIS
LIN {X 0.050,Y -425.520,Z 646.994,A 0.000,B 0.000,C 90.000,E1 34.978} C_DIS
LIN {X 0.084,Y -426.316,Z 646.985,A 0.000,B 0.000,C 90.000,E1 33.293} C_DIS
LIN {X 0.033,Y -426.935,Z 646.978,A 0.000,B 0.000,C 90.000,E1 31.957} C_DIS
LIN {X -0.013,Y -427.894,Z 646.966,A 0.000,B 0.000,C 90.000,E1 29.951} C_DIS
LIN {X -0.257,Y -428.869,Z 646.955,A 0.000,B 0.000,C 90.000,E1 27.975} C_DIS
LIN {X 0.080,Y -429.913,Z 646.944,A 0.000,B 0.000,C 90.000,E1 25.924} C_DIS
LIN {X -0.131,Y -431.911,Z 646.927,A 0.000,B 0.000,C 90.000,E1 22.950} C_DIS
LIN {X 0.145,Y -433.420,Z 646.916,A 0.000,B 0.000,C 90.000,E1 20.918} C_DIS
LIN {X 0.070,Y -434.540,Z 646.907,A 0.000,B 0.000,C 90.000,E1 19.268} C_DIS
LIN {X -0.069,Y -435.866,Z 646.894,A 0.000,B 0.000,C 90.000,E1 16.968} C_DIS
LIN {X 0.167,Y -437.193,Z 646.883,A 0.000,B 0.000,C 90.000,E1 14.954} C_DIS
LIN {X -0.087,Y -438.720,Z 646.872,A 0.000,B 0.000,C 90.000,E1 13.008} C_DIS
LIN {X -0.013,Y -440.990,Z 646.858,A 0.000,B 0.000,C 90.000,E1 10.366} C_DIS
LIN {X -0.113,Y -443.577,Z 646.843,A 0.000,B 0.000,C 90.000,E1 7.757} C_DIS
LIN {X -0.097,Y -445.741,Z 646.832,A 0.000,B 0.000,C 90.000,E1 5.796} C_DIS
LIN {X -0.077,Y -448.025,Z 646.821,A 0.000,B 0.000,C 90.000,E1 3.841} C_DIS
LIN {X -0.209,Y -450.099,Z 646.812,A 0.000,B 0.000,C 90.000,E1 2.236} C_DIS
LIN {X 0.000,Y -453.152,Z 646.800,A 0.000,B 0.000,C 90.000,E1 360.000} C_DIS
LIN {X -0.215,Y -457.467,Z 646.785,A 0.000,B 0.000,C 90.000,E1 357.249} C_DIS
LIN {X 0.054,Y -460.734,Z 646.774,A 0.000,B 0.000,C 90.000,E1 355.298} C_DIS
LIN {X -0.238,Y -464.683,Z 646.762,A 0.000,B 0.000,C 90.000,E1 353.109} C_DIS
LIN {X 0.160,Y -468.564,Z 646.749,A 0.000,B 0.000,C 90.000,E1 350.849} C_DIS
LIN {X 0.089,Y -471.271,Z 646.741,A 0.000,B 0.000,C 90.000,E1 349.285} C_DIS
LIN {X 0.244,Y -474.032,Z 646.732,A 0.000,B 0.000,C 90.000,E1 347.701} C_DIS
LIN {X -0.169,Y -477.389,Z 646.721,A 0.000,B 0.000,C 90.000,E1 345.880} C_DIS
LIN {X -0.245,Y -480.290,Z 646.713,A 0.000,B 0.000,C 90.000,E1 344.338} C_DIS
LIN {X 0.176,Y -484.424,Z 646.701,A 0.000,B 0.000,C 90.000,E1 342.127} C_DIS
LIN {X 0.049,Y -486.834,Z 646.694,A 0.000,B 0.000,C 90.000,E1 340.913} C_DIS
LIN {X 0.010,Y -490.488,Z 646.684,A 0.000,B 0.000,C 90.000,E1 339.082} C_DIS
LIN {X 0.148,Y -492.845,Z 646.677,A 0.000,B 0.000,C 90.000,E1 337.847} C_DIS
LIN {X -0.088,Y -495.525,Z 646.669,A 0.000,B 0.000,C 90.000,E1 336.357} C_DIS
LIN {X 0.061,Y -497.035,Z 646.664,A 0.000,B 0.000,C 90.000,E1 335.433} C_DIS
LIN {X -0.082,Y -499.994,Z 646.654,A 0.000,B 0.000,C 90.000,E1 333.640} C_DIS
LIN {X 0.144,Y -503.461,Z 646.642,A 0.000,B 0.000,C 90.000,E1 331.513} C_DIS
LIN {X -0.179,Y -507.473,Z 646.630,A 0.000,B 0.000,C 90.000,E1 329.459} C_DIS
LIN {X -0.227,Y -509.007,Z 646.627,A 0.000,B 0.000,C 90.000,E1 328.869} C_DIS
LIN {X 0.101,Y -510.173,Z 646.625,A 0.000,B 0.000,C 90.000,E1 328.535} C_DIS
LIN {X -0.185,Y -511.646,Z 646.623,A 0.000,B 0.000,C 90.000,E1 328.122} C_DIS
LIN {X -0.026,Y -513.694,Z 646.620,A 0.000,B 0.000,C 90.000,E1 327.661} C_DIS
LIN {X -0.222,Y -515.925,Z 646.618,A 0.000,B 0.000,C 90.000,E1 327.327} C_DIS
LIN {X 0.011,Y -516.920,Z 646.618,A 0.000,B 0.000,C 90.000,E1 327.168} C_DIS
LIN {X 0.034,Y -519.876,Z 646.616,A 0.000,B 0.000,C 90.000,E1 326.834} C_DIS
LIN {X 0.103,Y -524.959,Z 646.613,A 0.000,B 0.000,C 90.000,E1 326.342} C_DIS
LIN {X -0.196,Y -538.119,Z 646.607,A 0.000,B 0.000,C 90.000,E1 325.308} C_DIS
LIN {X -0.226,Y -546.880,Z 646.603,A 0.000,B 0.000,C 90.000,E1 324.609} C_DIS
LIN {X 0.143,Y -553.856,Z 646.600,A 0.000,B 0.000,C 90.000,E1 323.989} C_DIS
LIN {X 0.273,Y -563.595,Z 646.595,A 0.000,B 0.000,C 90.000,E1 323.130} C_DIS
LIN {X 0.060,Y -571.615,Z 646.591,A 0.000,B 0.000,C 90.000,E1 322.431} C_DIS
LIN {X -0.218,Y -587.731,Z 646.583,A 0.000,B 0.000,C 90.000,E1 320.964} C_DIS
LIN {X -0.018,Y -598.060,Z 646.578,A 0.000,B 0.000,C 90.000,E1 319.952} C_DIS
LIN {X 0.013,Y -605.407,Z 646.573,A 0.000,B 0.000,C 90.000,E1 319.218} C_DIS
LIN {X 0.184,Y -610.136,Z 646.571,A 0.000,B 0.000,C 90.000,E1 318.690} C_DIS
LIN {X 0.276,Y -614.575,Z 646.568,A 0.000,B 0.000,C 90.000,E1 318.162} C_DIS
LIN {X -0.274,Y -621.916,Z 646.563,A 0.000,B 0.000,C 90.000,E1 317.310} C_DIS
LIN {X 0.265,Y -626.760,Z 646.559,A 0.000,B 0.000,C 90.000,E1 316.620} C_DIS
LIN {X -0.110,Y -632.235,Z 646.555,A 0.000,B 0.000,C 90.000,E1 315.891} C_DIS
LIN {X 0.068,Y -636.601,Z 646.551,A 0.000,B 0.000,C 90.000,E1 315.243} C_DIS
LIN {X 0.122,Y -644.171,Z 646.545,A 0.000,B 0.000,C 90.000,E1 314.109} C_DIS
LIN {X 0.272,Y -652.186,Z 646.538,A 0.000,B 0.000,C 90.000,E1 312.852} C_DIS
LIN {X 0.134,Y -656.613,Z 646.534,A 0.000,B 0.000,C 90.000,E1 312.123} C_DIS
LIN {X 0.114,Y -659.537,Z 646.531,A 0.000,B 0.000,C 90.000,E1 311.634} C_DIS
LIN {X 0.063,Y -664.182,Z 646.527,A 0.000,B 0.000,C 90.000,E1 310.782} C_DIS
LIN {X 0.064,Y -667.256,Z 646.523,A 0.000,B 0.000,C 90.000,E1 310.172} C_DIS
LIN {X -0.383,Y -669.595,Z 646.521,A 0.000,B 0.000,C 90.000,E1 309.725} C_DIS
LIN {X 0.124,Y -672.789,Z 646.517,A 0.000,B 0.000,C 90.000,E1 308.955} C_DIS
LIN {X -0.181,Y -675.722,Z 646.513,A 0.000,B 0.000,C 90.000,E1 308.257} C_DIS
LIN {X -0.035,Y -678.359,Z 646.508,A 0.000,B 0.000,C 90.000,E1 307.523} C_DIS
LIN {X 0.133,Y -680.839,Z 646.505,A 0.000,B 0.000,C 90.000,E1 306.790} C_DIS
LIN {X -0.068,Y -683.854,Z 646.499,A 0.000,B 0.000,C 90.000,E1 305.851} C_DIS
LIN {X -0.053,Y -687.416,Z 646.493,A 0.000,B 0.000,C 90.000,E1 304.659} C_DIS
LIN {X 0.205,Y -690.688,Z 646.486,A 0.000,B 0.000,C 90.000,E1 303.452} C_DIS
LIN {X -0.276,Y -693.092,Z 646.481,A 0.000,B 0.000,C 90.000,E1 302.546} C_DIS
LIN {X -0.150,Y -695.312,Z 646.476,A 0.000,B 0.000,C 90.000,E1 301.592} C_DIS
LIN {X -0.360,Y -697.387,Z 646.470,A 0.000,B 0.000,C 90.000,E1 300.669} C_DIS
LIN {X 0.416,Y -699.292,Z 646.465,A 0.000,B 0.000,C 90.000,E1 299.667} C_DIS
LIN {X 0.259,Y -701.033,Z 646.460,A 0.000,B 0.000,C 90.000,E1 298.743} C_DIS
LIN {X -0.212,Y -702.565,Z 646.455,A 0.000,B 0.000,C 90.000,E1 297.847} C_DIS
LIN {X 0.289,Y -703.870,Z 646.449,A 0.000,B 0.000,C 90.000,E1 296.873} C_DIS
LIN {X 0.202,Y -704.683,Z 646.446,A 0.000,B 0.000,C 90.000,E1 296.181} C_DIS
LIN {X 0.144,Y -704.816,Z 646.443,A 0.000,B 0.000,C 90.000,E1 295.720} C_DIS
LIN {X 0.432,Y -704.723,Z 646.442,A 0.000,B 0.000,C 90.000,E1 295.463} C_DIS
LIN {X 0.068,Y -703.917,Z 646.439,A 0.000,B 0.000,C 90.000,E1 295.027} C_DIS
LIN {X 0.354,Y -703.159,Z 646.438,A 0.000,B 0.000,C 90.000,E1 294.771} C_DIS
LIN {X -0.016,Y -700.113,Z 646.435,A 0.000,B 0.000,C 90.000,E1 294.335} C_DIS
LIN {X 0.119,Y -699.248,Z 646.435,A 0.000,B 0.000,C 90.000,E1 294.207} C_DIS
LIN {X 0.255,Y -697.976,Z 646.434,A 0.000,B 0.000,C 90.000,E1 294.079} C_DIS
LIN {X -0.198,Y -696.044,Z 646.433,A 0.000,B 0.000,C 90.000,E1 294.003} C_DIS
LIN {X -0.242,Y -691.830,Z 646.432,A 0.000,B 0.000,C 90.000,E1 293.823} C_DIS
LIN {X 0.292,Y -688.029,Z 646.432,A 0.000,B 0.000,C 90.000,E1 293.643} C_DIS
LIN {X -0.018,Y -681.436,Z 646.431,A 0.000,B 0.000,C 90.000,E1 293.515} C_DIS
LIN {X 0.074,Y -670.515,Z 646.430,A 0.000,B 0.000,C 90.000,E1 293.387} C_DIS
LIN {X -0.200,Y -663.613,Z 646.430,A 0.000,B 0.000,C 90.000,E1 293.334} C_DIS
LIN {X -0.336,Y -652.970,Z 646.429,A 0.000,B 0.000,C 90.000,E1 293.206} C_DIS
LIN {X -0.047,Y -640.117,Z 646.428,A 0.000,B 0.000,C 90.000,E1 292.950} C_DIS
LIN {X 0.178,Y -630.047,Z 646.426,A 0.000,B 0.000,C 90.000,E1 292.717} C_DIS
LIN {X 0.282,Y -620.405,Z 646.425,A 0.000,B 0.000,C 90.000,E1 292.461} C_DIS
LIN {X 0.093,Y -593.054,Z 646.420,A 0.000,B 0.000,C 90.000,E1 291.663} C_DIS
LIN {X 0.159,Y -577.218,Z 646.418,A 0.000,B 0.000,C 90.000,E1 291.153} C_DIS
LIN {X 0.161,Y -563.224,Z 646.415,A 0.000,B 0.000,C 90.000,E1 290.737} C_DIS
LIN {X 0.220,Y -560.225,Z 646.415,A 0.000,B 0.000,C 90.000,E1 290.610} C_DIS
LIN {X -0.150,Y -556.785,Z 646.413,A 0.000,B 0.000,C 90.000,E1 290.429} C_DIS
LIN {X -0.199,Y -556.757,Z 646.413,A 0.000,B 0.000,C 90.000,E1 290.429} C_DIS
LIN {X 0.003,Y -555.996,Z 646.413,A 0.000,B 0.000,C 90.000,E1 290.248} C_DIS
LIN {X -0.263,Y -555.626,Z 646.411,A 0.000,B 0.000,C 90.000,E1 290.066} C_DIS
LIN {X 0.027,Y -555.324,Z 646.410,A 0.000,B 0.000,C 90.000,E1 289.758} C_DIS
LIN {X 0.171,Y -555.254,Z 646.402,A 0.000,B 0.000,C 90.000,E1 288.362} C_DIS
LIN {X 0.018,Y -554.996,Z 646.394,A 0.000,B 0.000,C 90.000,E1 286.985} C_DIS
LIN {X -0.140,Y -554.575,Z 646.387,A 0.000,B 0.000,C 90.000,E1 285.607} C_DIS
LIN {X 0.082,Y -553.964,Z 646.379,A 0.000,B 0.000,C 90.000,E1 284.189} C_DIS
LIN {X -0.002,Y -552.898,Z 646.368,A 0.000,B 0.000,C 90.000,E1 282.243} C_DIS
LIN {X 0.184,Y -552.092,Z 646.359,A 0.000,B 0.000,C 90.000,E1 280.546} C_DIS
LIN {X -0.039,Y -551.173,Z 646.345,A 0.000,B 0.000,C 90.000,E1 278.049} C_DIS
LIN {X 0.063,Y -550.492,Z 646.332,A 0.000,B 0.000,C 90.000,E1 275.796} C_DIS
LIN {X -0.016,Y -550.023,Z 646.321,A 0.000,B 0.000,C 90.000,E1 273.841} C_DIS
LIN {X 0.221,Y -549.788,Z 646.315,A 0.000,B 0.000,C 90.000,E1 272.694} C_DIS
LIN {X -0.097,Y -549.485,Z 646.309,A 0.000,B 0.000,C 90.000,E1 271.604} C_DIS
LIN {X 0.221,Y -548.833,Z 646.300,A 0.000,B 0.000,C 90.000,E1 269.885} C_DIS
LIN {X 0.037,Y -547.810,Z 646.289,A 0.000,B 0.000,C 90.000,E1 267.936} C_DIS
LIN {X -0.257,Y -547.150,Z 646.281,A 0.000,B 0.000,C 90.000,E1 266.560} C_DIS
LIN {X -0.064,Y -546.480,Z 646.275,A 0.000,B 0.000,C 90.000,E1 265.412} C_DIS
LIN {X -0.191,Y -545.008,Z 646.264,A 0.000,B 0.000,C 90.000,E1 263.451} C_DIS
LIN {X 0.012,Y -543.917,Z 646.257,A 0.000,B 0.000,C 90.000,E1 262.299} C_DIS
LIN {X -0.187,Y -542.334,Z 646.249,A 0.000,B 0.000,C 90.000,E1 260.905} C_DIS
LIN {X -0.177,Y -540.125,Z 646.237,A 0.000,B 0.000,C 90.000,E1 258.634} C_DIS
LIN {X 0.046,Y -539.367,Z 646.232,A 0.000,B 0.000,C 90.000,E1 257.757} C_DIS
LIN {X 0.182,Y -537.481,Z 646.219,A 0.000,B 0.000,C 90.000,E1 255.463} C_DIS
LIN {X 0.082,Y -536.177,Z 646.211,A 0.000,B 0.000,C 90.000,E1 254.047} C_DIS
LIN {X -0.214,Y -534.525,Z 646.202,A 0.000,B 0.000,C 90.000,E1 252.362} C_DIS
LIN {X -0.061,Y -533.206,Z 646.194,A 0.000,B 0.000,C 90.000,E1 250.913} C_DIS
LIN {X -0.147,Y -532.195,Z 646.189,A 0.000,B 0.000,C 90.000,E1 250.061} C_DIS
LIN {X -0.053,Y -530.614,Z 646.183,A 0.000,B 0.000,C 90.000,E1 248.901} C_DIS
LIN {X 0.212,Y -528.954,Z 646.176,A 0.000,B 0.000,C 90.000,E1 247.720} C_DIS
LIN {X -0.238,Y -527.164,Z 646.170,A 0.000,B 0.000,C 90.000,E1 246.613} C_DIS
LIN {X -0.123,Y -524.567,Z 646.162,A 0.000,B 0.000,C 90.000,E1 245.153} C_DIS
LIN {X 0.039,Y -522.316,Z 646.155,A 0.000,B 0.000,C 90.000,E1 243.973} C_DIS
LIN {X -0.036,Y -518.640,Z 646.146,A 0.000,B 0.000,C 90.000,E1 242.231} C_DIS
LIN {X -0.303,Y -515.574,Z 646.138,A 0.000,B 0.000,C 90.000,E1 240.795} C_DIS
LIN {X 0.070,Y -512.215,Z 646.129,A 0.000,B 0.000,C 90.000,E1 239.282} C_DIS
LIN {X 0.203,Y -508.786,Z 646.121,A 0.000,B 0.000,C 90.000,E1 237.788} C_DIS
LIN {X 0.169,Y -504.599,Z 646.111,A 0.000,B 0.000,C 90.000,E1 236.008} C_DIS
LIN {X 0.318,Y -499.979,Z 646.101,A 0.000,B 0.000,C 90.000,E1 234.196} C_DIS
LIN {X 0.116,Y -494.529,Z 646.090,A 0.000,B 0.000,C 90.000,E1 232.110} C_DIS
LIN {X 0.080,Y -490.828,Z 646.081,A 0.000,B 0.000,C 90.000,E1 230.598} C_DIS
LIN {X -0.125,Y -485.741,Z 646.069,A 0.000,B 0.000,C 90.000,E1 228.485} C_DIS
LIN {X 0.311,Y -479.901,Z 646.056,A 0.000,B 0.000,C 90.000,E1 225.972} C_DIS
LIN {X 0.000,Y -475.437,Z 646.045,A 0.000,B 0.000,C 90.000,E1 224.150} C_DIS
LIN {X -0.061,Y -471.057,Z 646.035,A 0.000,B 0.000,C 90.000,E1 222.285} C_DIS
LIN {X -0.104,Y -466.259,Z 646.023,A 0.000,B 0.000,C 90.000,E1 220.092} C_DIS
LIN {X -0.208,Y -461.554,Z 646.010,A 0.000,B 0.000,C 90.000,E1 217.890} C_DIS
LIN {X 0.127,Y -455.827,Z 645.994,A 0.000,B 0.000,C 90.000,E1 214.978} C_DIS
LIN {X 0.035,Y -453.479,Z 645.987,A 0.000,B 0.000,C 90.000,E1 213.706} C_DIS
LIN {X -0.092,Y -449.364,Z 645.975,A 0.000,B 0.000,C 90.000,E1 211.465} C_DIS
LIN {X 0.147,Y -447.679,Z 645.969,A 0.000,B 0.000,C 90.000,E1 210.463} C_DIS
LIN {X -0.115,Y -444.806,Z 645.960,A 0.000,B 0.000,C 90.000,E1 208.871} C_DIS
LIN {X 0.027,Y -440.661,Z 645.948,A 0.000,B 0.000,C 90.000,E1 206.565} C_DIS
LIN {X 0.201,Y -437.652,Z 645.939,A 0.000,B 0.000,C 90.000,E1 204.899} C_DIS
LIN {X -0.050,Y -434.003,Z 645.927,A 0.000,B 0.000,C 90.000,E1 202.950} C_DIS
LIN {X 0.207,Y -431.673,Z 645.920,A 0.000,B 0.000,C 90.000,E1 201.589} C_DIS
LIN {X 0.082,Y -428.785,Z 645.911,A 0.000,B 0.000,C 90.000,E1 199.939} C_DIS
LIN {X -0.103,Y -425.974,Z 645.902,A 0.000,B 0.000,C 90.000,E1 198.290} C_DIS
LIN {X 0.163,Y -422.090,Z 645.888,A 0.000,B 0.000,C 90.000,E1 195.898} C_DIS
LIN {X -0.117,Y -419.432,Z 645.879,A 0.000,B 0.000,C 90.000,E1 194.245} C_DIS
LIN {X 0.017,Y -416.225,Z 645.868,A 0.000,B 0.000,C 90.000,E1 192.187} C_DIS
LIN {X 0.031,Y -412.639,Z 645.854,A 0.000,B 0.000,C 90.000,E1 189.792} C_DIS
LIN {X -0.164,Y -409.651,Z 645.843,A 0.000,B 0.000,C 90.000,E1 187.757} C_DIS
LIN {X -0.129,Y -406.218,Z 645.830,A 0.000,B 0.000,C 90.000,E1 185.334} C_DIS
LIN {X 0.066,Y -402.381,Z 645.812,A 0.000,B 0.000,C 90.000,E1 182.178} C_DIS
LIN {X -0.037,Y -398.435,Z 645.789,A 0.000,B 0.000,C 90.000,E1 177.993} C_DIS
LIN {X -0.203,Y -396.150,Z 645.767,A 0.000,B 0.000,C 90.000,E1 174.147} C_DIS
LIN {X -0.079,Y -395.278,Z 645.754,A 0.000,B 0.000,C 90.000,E1 171.659} C_DIS
LIN {X 0.122,Y -394.888,Z 645.742,A 0.000,B 0.000,C 90.000,E1 169.511} C_DIS
LIN {X -0.040,Y -394.706,Z 645.724,A 0.000,B 0.000,C 90.000,E1 166.353} C_DIS
LIN {X 0.095,Y -394.793,Z 645.712,A 0.000,B 0.000,C 90.000,E1 164.212} C_DIS
LIN {X -0.147,Y -395.098,Z 645.701,A 0.000,B 0.000,C 90.000,E1 162.127} C_DIS
LIN {X -0.209,Y -395.424,Z 645.691,A 0.000,B 0.000,C 90.000,E1 160.369} C_DIS
LIN {X -0.066,Y -395.856,Z 645.679,A 0.000,B 0.000,C 90.000,E1 158.230} C_DIS
LIN {X 0.018,Y -396.403,Z 645.667,A 0.000,B 0.000,C 90.000,E1 156.102} C_DIS
LIN {X 0.115,Y -396.905,Z 645.656,A 0.000,B 0.000,C 90.000,E1 153.973} C_DIS
LIN {X -0.143,Y -397.414,Z 645.644,A 0.000,B 0.000,C 90.000,E1 151.897} C_DIS
LIN {X 0.152,Y -397.977,Z 645.632,A 0.000,B 0.000,C 90.000,E1 149.744} C_DIS
LIN {X 0.091,Y -398.467,Z 645.622,A 0.000,B 0.000,C 90.000,E1 147.995} C_DIS
LIN {X 0.137,Y -399.215,Z 645.611,A 0.000,B 0.000,C 90.000,E1 145.881} C_DIS
LIN {X 0.202,Y -400.226,Z 645.597,A 0.000,B 0.000,C 90.000,E1 143.417} C_DIS
LIN {X -0.024,Y -401.013,Z 645.587,A 0.000,B 0.000,C 90.000,E1 141.698} C_DIS
LIN {X 0.078,Y -401.932,Z 645.576,A 0.000,B 0.000,C 90.000,E1 139.585} C_DIS
LIN {X 0.086,Y -402.713,Z 645.566,A 0.000,B 0.000,C 90.000,E1 137.838} C_DIS
LIN {X 0.202,Y -403.623,Z 645.554,A 0.000,B 0.000,C 90.000,E1 135.729} C_DIS
LIN {X 0.158,Y -404.800,Z 645.541,A 0.000,B 0.000,C 90.000,E1 133.299} C_DIS
LIN {X -0.087,Y -405.839,Z 645.531,A 0.000,B 0.000,C 90.000,E1 131.595} C_DIS
LIN {X 0.163,Y -407.381,Z 645.523,A 0.000,B 0.000,C 90.000,E1 130.172} C_DIS
LIN {X 0.101,Y -408.951,Z 645.519,A 0.000,B 0.000,C 90.000,E1 129.402} C_DIS
LIN {X -0.129,Y -411.382,Z 645.516,A 0.000,B 0.000,C 90.000,E1 128.830} C_DIS
LIN {X -0.159,Y -413.065,Z 645.515,A 0.000,B 0.000,C 90.000,E1 128.624} C_DIS
LIN {X 0.090,Y -414.840,Z 645.513,A 0.000,B 0.000,C 90.000,E1 128.338} C_DIS
LIN {X 0.112,Y -419.089,Z 645.511,A 0.000,B 0.000,C 90.000,E1 127.935} C_DIS
LIN {X 0.042,Y -424.064,Z 645.509,A 0.000,B 0.000,C 90.000,E1 127.569} C_DIS
LIN {X -0.225,Y -446.931,Z 645.500,A 0.000,B 0.000,C 90.000,E1 126.091} C_DIS
LIN {X 0.057,Y -456.349,Z 645.497,A 0.000,B 0.000,C 90.000,E1 125.438} C_DIS
LIN {X -0.254,Y -465.812,Z 645.493,A 0.000,B 0.000,C 90.000,E1 124.818} C_DIS
LIN {X 0.202,Y -473.767,Z 645.490,A 0.000,B 0.000,C 90.000,E1 124.199} C_DIS
LIN {X -0.181,Y -479.925,Z 645.488,A 0.000,B 0.000,C 90.000,E1 123.785} C_DIS
LIN {X 0.129,Y -489.120,Z 645.484,A 0.000,B 0.000,C 90.000,E1 123.038} C_DIS
LIN {X 0.203,Y -495.047,Z 645.481,A 0.000,B 0.000,C 90.000,E1 122.546} C_DIS
LIN {X 0.245,Y -503.665,Z 645.477,A 0.000,B 0.000,C 90.000,E1 121.799} C_DIS
LIN {X 0.059,Y -510.566,Z 645.473,A 0.000,B 0.000,C 90.000,E1 121.209} C_DIS
LIN {X -0.248,Y -519.083,Z 645.469,A 0.000,B 0.000,C 90.000,E1 120.463} C_DIS
LIN {X 0.021,Y -528.040,Z 645.464,A 0.000,B 0.000,C 90.000,E1 119.539} C_DIS
LIN {X 0.091,Y -533.975,Z 645.461,A 0.000,B 0.000,C 90.000,E1 118.899} C_DIS
LIN {X -0.115,Y -538.789,Z 645.458,A 0.000,B 0.000,C 90.000,E1 118.359} C_DIS
LIN {X 0.073,Y -543.310,Z 645.454,A 0.000,B 0.000,C 90.000,E1 117.769} C_DIS
LIN {X 0.045,Y -547.333,Z 645.451,A 0.000,B 0.000,C 90.000,E1 117.206} C_DIS
LIN {X 0.181,Y -551.639,Z 645.447,A 0.000,B 0.000,C 90.000,E1 116.488} C_DIS
LIN {X 0.108,Y -555.488,Z 645.443,A 0.000,B 0.000,C 90.000,E1 115.796} C_DIS
LIN {X 0.204,Y -559.571,Z 645.439,A 0.000,B 0.000,C 90.000,E1 114.951} C_DIS
LIN {X 0.101,Y -563.239,Z 645.434,A 0.000,B 0.000,C 90.000,E1 114.131} C_DIS
LIN {X 0.136,Y -567.744,Z 645.428,A 0.000,B 0.000,C 90.000,E1 113.025} C_DIS
LIN {X 0.110,Y -570.889,Z 645.423,A 0.000,B 0.000,C 90.000,E1 112.206} C_DIS
LIN {X -0.102,Y -573.684,Z 645.419,A 0.000,B 0.000,C 90.000,E1 111.408} C_DIS
LIN {X -0.286,Y -576.145,Z 645.414,A 0.000,B 0.000,C 90.000,E1 110.610} C_DIS
LIN {X 0.098,Y -578.470,Z 645.410,A 0.000,B 0.000,C 90.000,E1 109.758} C_DIS
LIN {X 0.161,Y -581.256,Z 645.404,A 0.000,B 0.000,C 90.000,E1 108.671} C_DIS
LIN {X -0.292,Y -583.687,Z 645.398,A 0.000,B 0.000,C 90.000,E1 107.638} C_DIS
LIN {X 0.146,Y -587.799,Z 645.387,A 0.000,B 0.000,C 90.000,E1 105.717} C_DIS
LIN {X -0.153,Y -590.883,Z 645.380,A 0.000,B 0.000,C 90.000,E1 104.411} C_DIS
LIN {X -0.269,Y -594.589,Z 645.371,A 0.000,B 0.000,C 90.000,E1 102.827} C_DIS
LIN {X -0.011,Y -597.561,Z 645.364,A 0.000,B 0.000,C 90.000,E1 101.478} C_DIS
LIN {X -0.102,Y -601.062,Z 645.355,A 0.000,B 0.000,C 90.000,E1 99.905} C_DIS
LIN {X 0.154,Y -603.909,Z 645.348,A 0.000,B 0.000,C 90.000,E1 98.568} C_DIS
LIN {X 0.050,Y -606.005,Z 645.342,A 0.000,B 0.000,C 90.000,E1 97.530} C_DIS
LIN {X 0.051,Y -607.963,Z 645.336,A 0.000,B 0.000,C 90.000,E1 96.486} C_DIS
LIN {X 0.266,Y -610.142,Z 645.329,A 0.000,B 0.000,C 90.000,E1 95.163} C_DIS
LIN {X 0.197,Y -611.786,Z 645.323,A 0.000,B 0.000,C 90.000,E1 94.131} C_DIS
LIN {X -0.134,Y -613.604,Z 645.316,A 0.000,B 0.000,C 90.000,E1 92.865} C_DIS
LIN {X -0.180,Y -614.831,Z 645.310,A 0.000,B 0.000,C 90.000,E1 91.835} C_DIS
LIN {X 0.123,Y -615.595,Z 645.306,A 0.000,B 0.000,C 90.000,E1 91.031} C_DIS
LIN {X -0.200,Y -616.594,Z 645.299,A 0.000,B 0.000,C 90.000,E1 89.771} C_DIS
LIN {X -0.202,Y -617.125,Z 645.293,A 0.000,B 0.000,C 90.000,E1 88.740} C_DIS
LIN {X -0.180,Y -617.490,Z 645.287,A 0.000,B 0.000,C 90.000,E1 87.707} C_DIS
LIN {X -0.148,Y -617.522,Z 645.281,A 0.000,B 0.000,C 90.000,E1 86.674} C_DIS
LIN {X 0.195,Y -617.451,Z 645.277,A 0.000,B 0.000,C 90.000,E1 85.869} C_DIS
LIN {X 0.221,Y -617.197,Z 645.271,A 0.000,B 0.000,C 90.000,E1 84.837} C_DIS
LIN {X -0.281,Y -616.376,Z 645.263,A 0.000,B 0.000,C 90.000,E1 83.337} C_DIS
LIN {X 0.145,Y -615.500,Z 645.256,A 0.000,B 0.000,C 90.000,E1 82.008} C_DIS
LIN {X -0.060,Y -614.063,Z 645.249,A 0.000,B 0.000,C 90.000,E1 80.735} C_DIS
LIN {X 0.054,Y -612.766,Z 645.243,A 0.000,B 0.000,C 90.000,E1 79.690} C_DIS
LIN {X -0.107,Y -610.850,Z 645.236,A 0.000,B 0.000,C 90.000,E1 78.409} C_DIS
LIN {X 0.158,Y -608.307,Z 645.227,A 0.000,B 0.000,C 90.000,E1 76.825} C_DIS
LIN {X 0.190,Y -605.953,Z 645.220,A 0.000,B 0.000,C 90.000,E1 75.519} C_DIS
LIN {X -0.286,Y -603.969,Z 645.214,A 0.000,B 0.000,C 90.000,E1 74.519} C_DIS
LIN {X -0.052,Y -601.800,Z 645.208,A 0.000,B 0.000,C 90.000,E1 73.449} C_DIS
LIN {X 0.037,Y -598.948,Z 645.201,A 0.000,B 0.000,C 90.000,E1 72.127} C_DIS
LIN {X -0.190,Y -596.455,Z 645.195,A 0.000,B 0.000,C 90.000,E1 71.094} C_DIS
LIN {X 0.112,Y -593.630,Z 645.189,A 0.000,B 0.000,C 90.000,E1 70.007} C_DIS
LIN {X 0.021,Y -590.442,Z 645.183,A 0.000,B 0.000,C 90.000,E1 68.954} C_DIS
LIN {X 0.013,Y -587.791,Z 645.179,A 0.000,B 0.000,C 90.000,E1 68.156} C_DIS
LIN {X -0.150,Y -583.867,Z 645.173,A 0.000,B 0.000,C 90.000,E1 67.102} C_DIS
LIN {X -0.234,Y -580.732,Z 645.168,A 0.000,B 0.000,C 90.000,E1 66.305} C_DIS
LIN {X -0.264,Y -576.147,Z 645.162,A 0.000,B 0.000,C 90.000,E1 65.229} C_DIS
LIN {X -0.119,Y -573.146,Z 645.159,A 0.000,B 0.000,C 90.000,E1 64.537} C_DIS
LIN {X -0.092,Y -569.162,Z 645.154,A 0.000,B 0.000,C 90.000,E1 63.717} C_DIS
LIN {X -0.183,Y -566.364,Z 645.151,A 0.000,B 0.000,C 90.000,E1 63.179} C_DIS
LIN {X -0.231,Y -561.621,Z 645.146,A 0.000,B 0.000,C 90.000,E1 62.359} C_DIS
LIN {X 0.131,Y -558.217,Z 645.143,A 0.000,B 0.000,C 90.000,E1 61.769} C_DIS
LIN {X -0.214,Y -554.505,Z 645.140,A 0.000,B 0.000,C 90.000,E1 61.257} C_DIS
LIN {X -0.230,Y -550.408,Z 645.137,A 0.000,B 0.000,C 90.000,E1 60.717} C_DIS
LIN {X -0.065,Y -544.932,Z 645.134,A 0.000,B 0.000,C 90.000,E1 60.049} C_DIS
LIN {X 0.062,Y -540.204,Z 645.131,A 0.000,B 0.000,C 90.000,E1 59.537} C_DIS
LIN {X -0.048,Y -536.023,Z 645.129,A 0.000,B 0.000,C 90.000,E1 59.154} C_DIS
LIN {X -0.044,Y -531.592,Z 645.127,A 0.000,B 0.000,C 90.000,E1 58.791} C_DIS
LIN {X 0.202,Y -524.258,Z 645.124,A 0.000,B 0.000,C 90.000,E1 58.201} C_DIS
LIN {X -0.170,Y -519.273,Z 645.122,A 0.000,B 0.000,C 90.000,E1 57.916} C_DIS
LIN {X -0.055,Y -512.585,Z 645.119,A 0.000,B 0.000,C 90.000,E1 57.502} C_DIS
LIN {X -0.287,Y -507.634,Z 645.118,A 0.000,B 0.000,C 90.000,E1 57.248} C_DIS
LIN {X 0.106,Y -491.028,Z 645.113,A 0.000,B 0.000,C 90.000,E1 56.342} C_DIS
LIN {X -0.082,Y -479.171,Z 645.110,A 0.000,B 0.000,C 90.000,E1 55.754} C_DIS
LIN {X 0.033,Y -460.731,Z 645.104,A 0.000,B 0.000,C 90.000,E1 54.769} C_DIS
LIN {X -0.163,Y -442.334,Z 645.099,A 0.000,B 0.000,C 90.000,E1 53.783} C_DIS
LIN {X 0.115,Y -436.684,Z 645.097,A 0.000,B 0.000,C 90.000,E1 53.417} C_DIS
LIN {X 0.072,Y -436.612,Z 645.097,A 0.000,B 0.000,C 90.000,E1 53.417} C_DIS
LIN {X 0.184,Y -431.354,Z 645.082,A 0.000,B 0.000,C 90.000,E1 50.723} C_DIS
LIN {X -0.073,Y -422.484,Z 645.061,A 0.000,B 0.000,C 90.000,E1 46.905} C_DIS
LIN {X -0.097,Y -422.371,Z 645.060,A 0.000,B 0.000,C 90.000,E1 46.824} C_DIS
LIN {X -0.120,Y -422.649,Z 645.054,A 0.000,B 0.000,C 90.000,E1 45.729} C_DIS
LIN {X 0.177,Y -422.793,Z 645.048,A 0.000,B 0.000,C 90.000,E1 44.676} C_DIS
LIN {X 0.094,Y -423.134,Z 645.035,A 0.000,B 0.000,C 90.000,E1 42.324} C_DIS
LIN {X 0.058,Y -423.826,Z 645.022,A 0.000,B 0.000,C 90.000,E1 39.967} C_DIS
LIN {X -0.021,Y -424.979,Z 645.007,A 0.000,B 0.000,C 90.000,E1 37.282} C_DIS
LIN {X -0.148,Y -426.156,Z 644.994,A 0.000,B 0.000,C 90.000,E1 34.945} C_DIS
LIN {X 0.219,Y -427.236,Z 644.981,A 0.000,B 0.000,C 90.000,E1 32.546} C_DIS
LIN {X -0.187,Y -428.039,Z 644.972,A 0.000,B 0.000,C 90.000,E1 30.924} C_DIS
LIN {X 0.154,Y -428.785,Z 644.962,A 0.000,B 0.000,C 90.000,E1 29.205} C_DIS
LIN {X 0.102,Y -429.735,Z 644.951,A 0.000,B 0.000,C 90.000,E1 27.206} C_DIS
LIN {X 0.079,Y -430.627,Z 644.942,A 0.000,B 0.000,C 90.000,E1 25.540} C_DIS
LIN {X -0.099,Y -432.388,Z 644.927,A 0.000,B 0.000,C 90.000,E1 22.898} C_DIS
LIN {X -0.034,Y -433.604,Z 644.918,A 0.000,B 0.000,C 90.000,E1 21.227} C_DIS
LIN {X 0.132,Y -434.925,Z 644.907,A 0.000,B 0.000,C 90.000,E1 19.214} C_DIS
LIN {X 0.185,Y -436.046,Z 644.896,A 0.000,B 0.000,C 90.000,E1 17.221} C_DIS
LIN {X -0.165,Y -437.554,Z 644.883,A 0.000,B 0.000,C 90.000,E1 14.954} C_DIS
LIN {X 0.115,Y -439.085,Z 644.872,A 0.000,B 0.000,C 90.000,E1 12.939} C_DIS
LIN {X 0.107,Y -441.329,Z 644.857,A 0.000,B 0.000,C 90.000,E1 10.310} C_DIS
LIN {X 0.020,Y -443.888,Z 644.843,A 0.000,B 0.000,C 90.000,E1 7.701} C_DIS
LIN {X 0.045,Y -446.009,Z 644.832,A 0.000,B 0.000,C 90.000,E1 5.739} C_DIS
LIN {X 0.218,Y -448.679,Z 644.819,A 0.000,B 0.000,C 90.000,E1 3.440} C_DIS
LIN {X 0.106,Y -450.758,Z 644.810,A 0.000,B 0.000,C 90.000,E1 1.835} C_DIS
LIN {X 0.000,Y -453.313,Z 644.800,A 0.000,B 0.000,C 90.000,E1 360.000} C_DIS
LIN {X -0.210,Y -457.609,Z 644.785,A 0.000,B 0.000,C 90.000,E1 357.249} C_DIS
LIN {X 0.061,Y -460.854,Z 644.774,A 0.000,B 0.000,C 90.000,E1 355.298} C_DIS
LIN {X -0.228,Y -464.780,Z 644.762,A 0.000,B 0.000,C 90.000,E1 353.109} C_DIS
LIN {X 0.174,Y -468.632,Z 644.749,A 0.000,B 0.000,C 90.000,E1 350.849} C_DIS
LIN {X -0.179,Y -470.822,Z 644.742,A 0.000,B 0.000,C 90.000,E1 349.634} C_DIS
LIN {X -0.203,Y -474.096,Z 644.732,A 0.000,B 0.000,C 90.000,E1 347.757} C_DIS
LIN {X -0.149,Y -477.453,Z 644.721,A 0.000,B 0.000,C 90.000,E1 345.880} C_DIS
LIN {X -0.225,Y -480.356,Z 644.713,A 0.000,B 0.000,C 90.000,E1 344.338} C_DIS
LIN {X 0.200,Y -484.489,Z 644.701,A 0.000,B 0.000,C 90.000,E1 342.127} C_DIS
LIN {X 0.072,Y -486.899,Z 644.694,A 0.000,B 0.000,C 90.000,E1 340.913} C_DIS
LIN {X 0.065,Y -491.142,Z 644.682,A 0.000,B 0.000,C 90.000,E1 338.773} C_DIS
LIN {X 0.214,Y -493.446,Z 644.675,A 0.000,B 0.000,C 90.000,E1 337.539} C_DIS
LIN {X -0.012,Y -496.065,Z 644.667,A 0.000,B 0.000,C 90.000,E1 336.049} C_DIS
LIN {X -0.048,Y -497.998,Z 644.660,A 0.000,B 0.000,C 90.000,E1 334.845} C_DIS
LIN {X 0.004,Y -500.475,Z 644.652,A 0.000,B 0.000,C 90.000,E1 333.332} C_DIS
LIN {X 0.095,Y -504.419,Z 644.639,A 0.000,B 0.000,C 90.000,E1 330.923} C_DIS
LIN {X 0.169,Y -507.932,Z 644.629,A 0.000,B 0.000,C 90.000,E1 329.125} C_DIS
LIN {X 0.020,Y -510.404,Z 644.624,A 0.000,B 0.000,C 90.000,E1 328.250} C_DIS
LIN {X -0.164,Y -510.890,Z 644.623,A 0.000,B 0.000,C 90.000,E1 328.122} C_DIS
LIN {X -0.194,Y -513.383,Z 644.620,A 0.000,B 0.000,C 90.000,E1 327.533} C_DIS
LIN {X 0.251,Y -515.872,Z 644.617,A 0.000,B 0.000,C 90.000,E1 327.041} C_DIS
LIN {X 0.182,Y -517.403,Z 644.616,A 0.000,B 0.000,C 90.000,E1 326.834} C_DIS
LIN {X 0.111,Y -519.884,Z 644.614,A 0.000,B 0.000,C 90.000,E1 326.548} C_DIS
LIN {X -0.239,Y -522.809,Z 644.613,A 0.000,B 0.000,C 90.000,E1 326.294} C_DIS
LIN {X 0.017,Y -528.594,Z 644.610,A 0.000,B 0.000,C 90.000,E1 325.754} C_DIS
LIN {X 0.158,Y -544.267,Z 644.603,A 0.000,B 0.000,C 90.000,E1 324.482} C_DIS
LIN {X 0.003,Y -551.431,Z 644.600,A 0.000,B 0.000,C 90.000,E1 323.909} C_DIS
LIN {X -0.245,Y -559.881,Z 644.596,A 0.000,B 0.000,C 90.000,E1 323.210} C_DIS
LIN {X -0.178,Y -568.176,Z 644.591,A 0.000,B 0.000,C 90.000,E1 322.477} C_DIS
LIN {X 0.088,Y -580.322,Z 644.585,A 0.000,B 0.000,C 90.000,E1 321.331} C_DIS
LIN {X 0.021,Y -588.344,Z 644.581,A 0.000,B 0.000,C 90.000,E1 320.598} C_DIS
LIN {X 0.326,Y -596.189,Z 644.577,A 0.000,B 0.000,C 90.000,E1 319.828} C_DIS
LIN {X 0.170,Y -603.828,Z 644.573,A 0.000,B 0.000,C 90.000,E1 319.094} C_DIS
LIN {X -0.045,Y -607.496,Z 644.571,A 0.000,B 0.000,C 90.000,E1 318.728} C_DIS
LIN {X -0.019,Y -611.834,Z 644.568,A 0.000,B 0.000,C 90.000,E1 318.243} C_DIS
LIN {X -0.342,Y -619.264,Z 644.563,A 0.000,B 0.000,C 90.000,E1 317.391} C_DIS
LIN {X -0.179,Y -625.165,Z 644.559,A 0.000,B 0.000,C 90.000,E1 316.620} C_DIS
LIN {X -0.186,Y -631.653,Z 644.554,A 0.000,B 0.000,C 90.000,E1 315.729} C_DIS
LIN {X -0.113,Y -637.840,Z 644.549,A 0.000,B 0.000,C 90.000,E1 314.838} C_DIS
LIN {X 0.003,Y -644.579,Z 644.544,A 0.000,B 0.000,C 90.000,E1 313.824} C_DIS
LIN {X -0.260,Y -651.107,Z 644.538,A 0.000,B 0.000,C 90.000,E1 312.852} C_DIS
LIN {X 0.029,Y -656.423,Z 644.533,A 0.000,B 0.000,C 90.000,E1 311.962} C_DIS
LIN {X -0.036,Y -660.095,Z 644.530,A 0.000,B 0.000,C 90.000,E1 311.353} C_DIS
LIN {X -0.048,Y -664.042,Z 644.526,A 0.000,B 0.000,C 90.000,E1 310.620} C_DIS
LIN {X -0.014,Y -667.704,Z 644.522,A 0.000,B 0.000,C 90.000,E1 309.886} C_DIS
LIN {X 0.006,Y -671.631,Z 644.517,A 0.000,B 0.000,C 90.000,E1 309.036} C_DIS
LIN {X 0.106,Y -673.700,Z 644.514,A 0.000,B 0.000,C 90.000,E1 308.543} C_DIS
LIN {X -0.174,Y -677.352,Z 644.509,A 0.000,B 0.000,C 90.000,E1 307.604} C_DIS
LIN {X -0.015,Y -679.888,Z 644.505,A 0.000,B 0.000,C 90.000,E1 306.870} C_DIS
LIN {X -0.224,Y -683.003,Z 644.500,A 0.000,B 0.000,C 90.000,E1 305.931} C_DIS
LIN {X -0.222,Y -686.600,Z 644.493,A 0.000,B 0.000,C 90.000,E1 304.739} C_DIS
LIN {X -0.183,Y -689.322,Z 644.488,A 0.000,B 0.000,C 90.000,E1 303.785} C_DIS
LIN {X -0.101,Y -691.856,Z 644.482,A 0.000,B 0.000,C 90.000,E1 302.832} C_DIS
LIN {X 0.013,Y -694.206,Z 644.477,A 0.000,B 0.000,C 90.000,E1 301.878} C_DIS
LIN {X -0.198,Y -696.870,Z 644.471,A 0.000,B 0.000,C 90.000,E1 300.718} C_DIS
LIN {X 0.219,Y -698.886,Z 644.465,A 0.000,B 0.000,C 90.000,E1 299.745} C_DIS
LIN {X -0.283,Y -701.128,Z 644.459,A 0.000,B 0.000,C 90.000,E1 298.615} C_DIS
LIN {X 0.197,Y -702.663,Z 644.454,A 0.000,B 0.000,C 90.000,E1 297.641} C_DIS
LIN {X 0.093,Y -703.701,Z 644.450,A 0.000,B 0.000,C 90.000,E1 296.950} C_DIS
LIN {X 0.319,Y -704.560,Z 644.446,A 0.000,B 0.000,C 90.000,E1 296.232} C_DIS
LIN {X 0.241,Y -704.756,Z 644.442,A 0.000,B 0.000,C 90.000,E1 295.540} C_DIS
LIN {X 0.178,Y -703.933,Z 644.439,A 0.000,B 0.000,C 90.000,E1 295.079} C_DIS
LIN {X 0.167,Y -703.297,Z 644.438,A 0.000,B 0.000,C 90.000,E1 294.847} C_DIS
LIN {X -0.188,Y -701.881,Z 644.437,A 0.000,B 0.000,C 90.000,E1 294.643} C_DIS
LIN {X 0.226,Y -699.507,Z 644.435,A 0.000,B 0.000,C 90.000,E1 294.259} C_DIS
LIN {X 0.075,Y -698.448,Z 644.434,A 0.000,B 0.000,C 90.000,E1 294.155} C_DIS
LIN {X 0.209,Y -696.841,Z 644.434,A 0.000,B 0.000,C 90.000,E1 294.027} C_DIS
LIN {X 0.355,Y -692.600,Z 644.433,A 0.000,B 0.000,C 90.000,E1 293.823} C_DIS
LIN {X 0.089,Y -690.777,Z 644.432,A 0.000,B 0.000,C 90.000,E1 293.770} C_DIS
LIN {X 0.005,Y -686.500,Z 644.431,A 0.000,B 0.000,C 90.000,E1 293.643} C_DIS
LIN {X 0.272,Y -681.803,Z 644.431,A 0.000,B 0.000,C 90.000,E1 293.515} C_DIS
LIN {X -0.174,Y -679.450,Z 644.431,A 0.000,B 0.000,C 90.000,E1 293.515} C_DIS
LIN {X 0.071,Y -664.266,Z 644.430,A 0.000,B 0.000,C 90.000,E1 293.334} C_DIS
LIN {X 0.025,Y -650.899,Z 644.429,A 0.000,B 0.000,C 90.000,E1 293.153} C_DIS
LIN {X 0.155,Y -637.561,Z 644.427,A 0.000,B 0.000,C 90.000,E1 292.898} C_DIS
LIN {X 0.075,Y -628.179,Z 644.426,A 0.000,B 0.000,C 90.000,E1 292.695} C_DIS
LIN {X 0.088,Y -614.650,Z 644.424,A 0.000,B 0.000,C 90.000,E1 292.333} C_DIS
LIN {X 0.015,Y -578.688,Z 644.418,A 0.000,B 0.000,C 90.000,E1 291.227} C_DIS
LIN {X 0.199,Y -564.425,Z 644.416,A 0.000,B 0.000,C 90.000,E1 290.791} C_DIS
LIN {X 0.033,Y -559.647,Z 644.415,A 0.000,B 0.000,C 90.000,E1 290.610} C_DIS
LIN {X -0.116,Y -556.700,Z 644.413,A 0.000,B 0.000,C 90.000,E1 290.429} C_DIS
LIN {X -0.167,Y -556.670,Z 644.413,A 0.000,B 0.000,C 90.000,E1 290.429} C_DIS
LIN {X -0.118,Y -555.922,Z 644.412,A 0.000,B 0.000,C 90.000,E1 290.248} C_DIS
LIN {X 0.059,Y -555.425,Z 644.410,A 0.000,B 0.000,C 90.000,E1 289.812} C_DIS
LIN {X 0.077,Y -555.351,Z 644.402,A 0.000,B 0.000,C 90.000,E1 288.417} C_DIS
LIN {X -0.078,Y -555.103,Z 644.395,A 0.000,B 0.000,C 90.000,E1 287.040} C_DIS
LIN {X 0.177,Y -554.802,Z 644.388,A 0.000,B 0.000,C 90.000,E1 285.898} C_DIS
LIN {X -0.141,Y -554.216,Z 644.381,A 0.000,B 0.000,C 90.000,E1 284.537} C_DIS
LIN {X -0.053,Y -553.614,Z 644.375,A 0.000,B 0.000,C 90.000,E1 283.411} C_DIS
LIN {X 0.143,Y -552.741,Z 644.365,A 0.000,B 0.000,C 90.000,E1 281.715} C_DIS
LIN {X -0.223,Y -551.964,Z 644.356,A 0.000,B 0.000,C 90.000,E1 280.074} C_DIS
LIN {X -0.139,Y -551.288,Z 644.345,A 0.000,B 0.000,C 90.000,E1 278.106} C_DIS
LIN {X -0.036,Y -550.565,Z 644.333,A 0.000,B 0.000,C 90.000,E1 275.853} C_DIS
LIN {X -0.114,Y -550.095,Z 644.322,A 0.000,B 0.000,C 90.000,E1 273.898} C_DIS
LIN {X 0.123,Y -549.834,Z 644.315,A 0.000,B 0.000,C 90.000,E1 272.751} C_DIS
LIN {X -0.195,Y -549.535,Z 644.309,A 0.000,B 0.000,C 90.000,E1 271.661} C_DIS
LIN {X 0.123,Y -548.909,Z 644.300,A 0.000,B 0.000,C 90.000,E1 269.943} C_DIS
LIN {X -0.123,Y -548.017,Z 644.290,A 0.000,B 0.000,C 90.000,E1 268.282} C_DIS
LIN {X 0.123,Y -547.395,Z 644.283,A 0.000,B 0.000,C 90.000,E1 266.849} C_DIS
LIN {X -0.191,Y -546.773,Z 644.276,A 0.000,B 0.000,C 90.000,E1 265.755} C_DIS
LIN {X 0.073,Y -545.742,Z 644.269,A 0.000,B 0.000,C 90.000,E1 264.318} C_DIS
LIN {X -0.254,Y -544.886,Z 644.262,A 0.000,B 0.000,C 90.000,E1 263.223} C_DIS
LIN {X -0.069,Y -544.090,Z 644.258,A 0.000,B 0.000,C 90.000,E1 262.356} C_DIS
LIN {X 0.187,Y -542.509,Z 644.250,A 0.000,B 0.000,C 90.000,E1 260.914} C_DIS
LIN {X 0.286,Y -540.293,Z 644.237,A 0.000,B 0.000,C 90.000,E1 258.634} C_DIS
LIN {X 0.263,Y -538.518,Z 644.226,A 0.000,B 0.000,C 90.000,E1 256.645} C_DIS
LIN {X 0.189,Y -537.406,Z 644.218,A 0.000,B 0.000,C 90.000,E1 255.227} C_DIS
LIN {X -0.231,Y -535.791,Z 644.209,A 0.000,B 0.000,C 90.000,E1 253.559} C_DIS
LIN {X 0.211,Y -533.626,Z 644.196,A 0.000,B 0.000,C 90.000,E1 251.221} C_DIS
LIN {X 0.127,Y -532.727,Z 644.191,A 0.000,B 0.000,C 90.000,E1 250.369} C_DIS
LIN {X 0.227,Y -531.169,Z 644.185,A 0.000,B 0.000,C 90.000,E1 249.209} C_DIS
LIN {X -0.005,Y -529.112,Z 644.177,A 0.000,B 0.000,C 90.000,E1 247.794} C_DIS
LIN {X 0.057,Y -527.755,Z 644.172,A 0.000,B 0.000,C 90.000,E1 246.922} C_DIS
LIN {X -0.204,Y -525.814,Z 644.165,A 0.000,B 0.000,C 90.000,E1 245.793} C_DIS
LIN {X 0.204,Y -523.593,Z 644.159,A 0.000,B 0.000,C 90.000,E1 244.588} C_DIS
LIN {X -0.272,Y -521.832,Z 644.154,A 0.000,B 0.000,C 90.000,E1 243.768} C_DIS
LIN {X 0.109,Y -518.165,Z 644.144,A 0.000,B 0.000,C 90.000,E1 241.975} C_DIS
LIN {X -0.170,Y -515.054,Z 644.136,A 0.000,B 0.000,C 90.000,E1 240.539} C_DIS
LIN {X -0.250,Y -511.653,Z 644.128,A 0.000,B 0.000,C 90.000,E1 239.076} C_DIS
LIN {X -0.123,Y -508.170,Z 644.120,A 0.000,B 0.000,C 90.000,E1 237.582} C_DIS
LIN {X -0.062,Y -504.672,Z 644.112,A 0.000,B 0.000,C 90.000,E1 236.087} C_DIS
LIN {X -0.202,Y -500.824,Z 644.103,A 0.000,B 0.000,C 90.000,E1 234.609} C_DIS
LIN {X 0.157,Y -496.117,Z 644.093,A 0.000,B 0.000,C 90.000,E1 232.763} C_DIS
LIN {X 0.163,Y -490.892,Z 644.081,A 0.000,B 0.000,C 90.000,E1 230.642} C_DIS
LIN {X -0.030,Y -485.772,Z 644.070,A 0.000,B 0.000,C 90.000,E1 228.528} C_DIS
LIN {X -0.041,Y -480.625,Z 644.058,A 0.000,B 0.000,C 90.000,E1 226.377} C_DIS
LIN {X -0.222,Y -477.650,Z 644.051,A 0.000,B 0.000,C 90.000,E1 225.162} C_DIS
LIN {X 0.226,Y -474.672,Z 644.044,A 0.000,B 0.000,C 90.000,E1 223.866} C_DIS
LIN {X 0.069,Y -471.081,Z 644.035,A 0.000,B 0.000,C 90.000,E1 222.324} C_DIS
LIN {X -0.018,Y -466.277,Z 644.023,A 0.000,B 0.000,C 90.000,E1 220.135} C_DIS
LIN {X -0.170,Y -462.221,Z 644.012,A 0.000,B 0.000,C 90.000,E1 218.257} C_DIS
LIN {X -0.180,Y -456.426,Z 643.997,A 0.000,B 0.000,C 90.000,E1 215.391} C_DIS
LIN {X -0.163,Y -453.500,Z 643.988,A 0.000,B 0.000,C 90.000,E1 213.785} C_DIS
LIN {X 0.032,Y -448.805,Z 643.973,A 0.000,B 0.000,C 90.000,E1 211.180} C_DIS
LIN {X 0.177,Y -445.942,Z 643.964,A 0.000,B 0.000,C 90.000,E1 209.539} C_DIS
LIN {X 0.213,Y -443.629,Z 643.957,A 0.000,B 0.000,C 90.000,E1 208.231} C_DIS
LIN {X 0.091,Y -440.062,Z 643.946,A 0.000,B 0.000,C 90.000,E1 206.283} C_DIS
LIN {X 0.036,Y -437.655,Z 643.939,A 0.000,B 0.000,C 90.000,E1 204.975} C_DIS
LIN {X 0.189,Y -433.469,Z 643.926,A 0.000,B 0.000,C 90.000,E1 202.642} C_DIS
LIN {X 0.252,Y -430.527,Z 643.917,A 0.000,B 0.000,C 90.000,E1 200.972} C_DIS
LIN {X 0.088,Y -428.820,Z 643.911,A 0.000,B 0.000,C 90.000,E1 199.993} C_DIS
LIN {X -0.234,Y -426.030,Z 643.902,A 0.000,B 0.000,C 90.000,E1 198.362} C_DIS
LIN {X -0.180,Y -421.646,Z 643.887,A 0.000,B 0.000,C 90.000,E1 195.662} C_DIS
LIN {X 0.042,Y -418.969,Z 643.878,A 0.000,B 0.000,C 90.000,E1 193.939} C_DIS
LIN {X 0.066,Y -415.773,Z 643.866,A 0.000,B 0.000,C 90.000,E1 191.895} C_DIS
LIN {X 0.026,Y -412.718,Z 643.855,A 0.000,B 0.000,C 90.000,E1 189.849} C_DIS
LIN {X -0.198,Y -410.256,Z 643.845,A 0.000,B 0.000,C 90.000,E1 188.163} C_DIS
LIN {X -0.133,Y -406.299,Z 643.830,A 0.000,B 0.000,C 90.000,E1 185.391} C_DIS
LIN {X 0.099,Y -402.889,Z 643.814,A 0.000,B 0.000,C 90.000,E1 182.579} C_DIS
LIN {X 0.004,Y -398.791,Z 643.791,A 0.000,B 0.000,C 90.000,E1 178.396} C_DIS
LIN {X -0.125,Y -396.396,Z 643.770,A 0.000,B 0.000,C 90.000,E1 174.546} C_DIS
LIN {X -0.123,Y -395.420,Z 643.754,A 0.000,B 0.000,C 90.000,E1 171.724} C_DIS
LIN {X 0.107,Y -394.974,Z 643.740,A 0.000,B 0.000,C 90.000,E1 169.218} C_DIS
LIN {X -0.012,Y -394.825,Z 643.725,A 0.000,B 0.000,C 90.000,E1 166.408} C_DIS
LIN {X 0.070,Y -394.908,Z 643.715,A 0.000,B 0.000,C 90.000,E1 164.629} C_DIS
LIN {X -0.167,Y -395.189,Z 643.703,A 0.000,B 0.000,C 90.000,E1 162.543} C_DIS
LIN {X 0.150,Y -395.536,Z 643.693,A 0.000,B 0.000,C 90.000,E1 160.732} C_DIS
LIN {X -0.070,Y -395.939,Z 643.681,A 0.000,B 0.000,C 90.000,E1 158.646} C_DIS
LIN {X -0.073,Y -396.592,Z 643.668,A 0.000,B 0.000,C 90.000,E1 156.177} C_DIS
LIN {X 0.194,Y -397.092,Z 643.656,A 0.000,B 0.000,C 90.000,E1 154.024} C_DIS
LIN {X -0.053,Y -397.607,Z 643.644,A 0.000,B 0.000,C 90.000,E1 151.948} C_DIS
LIN {X 0.055,Y -398.208,Z 643.632,A 0.000,B 0.000,C 90.000,E1 149.822} C_DIS
LIN {X 0.086,Y -398.797,Z 643.621,A 0.000,B 0.000,C 90.000,E1 147.709} C_DIS
LIN {X 0.023,Y -399.702,Z 643.607,A 0.000,B 0.000,C 90.000,E1 145.261} C_DIS
LIN {X -0.223,Y -400.739,Z 643.593,A 0.000,B 0.000,C 90.000,E1 142.844} C_DIS
LIN {X -0.192,Y -401.491,Z 643.584,A 0.000,B 0.000,C 90.000,E1 141.090} C_DIS
LIN {X -0.013,Y -402.100,Z 643.576,A 0.000,B 0.000,C 90.000,E1 139.666} C_DIS
LIN {X -0.004,Y -402.826,Z 643.566,A 0.000,B 0.000,C 90.000,E1 137.919} C_DIS
LIN {X 0.114,Y -403.683,Z 643.555,A 0.000,B 0.000,C 90.000,E1 135.810} C_DIS
LIN {X 0.072,Y -404.831,Z 643.541,A 0.000,B 0.000,C 90.000,E1 133.380} C_DIS
LIN {X -0.036,Y -406.052,Z 643.530,A 0.000,B 0.000,C 90.000,E1 131.310} C_DIS
LIN {X 0.078,Y -407.146,Z 643.524,A 0.000,B 0.000,C 90.000,E1 130.253} C_DIS
LIN {X -0.090,Y -407.684,Z 643.522,A 0.000,B 0.000,C 90.000,E1 129.930} C_DIS
LIN {X 0.056,Y -408.391,Z 643.520,A 0.000,B 0.000,C 90.000,E1 129.564} C_DIS
LIN {X 0.205,Y -408.952,Z 643.518,A 0.000,B 0.000,C 90.000,E1 129.197} C_DIS
LIN {X 0.019,Y -410.815,Z 643.515,A 0.000,B 0.000,C 90.000,E1 128.705} C_DIS
LIN {X 0.142,Y -413.489,Z 643.513,A 0.000,B 0.000,C 90.000,E1 128.257} C_DIS
LIN {X -0.083,Y -418.211,Z 643.510,A 0.000,B 0.000,C 90.000,E1 127.810} C_DIS
LIN {X 0.024,Y -423.952,Z 643.508,A 0.000,B 0.000,C 90.000,E1 127.363} C_DIS
LIN {X -0.009,Y -449.876,Z 643.498,A 0.000,B 0.000,C 90.000,E1 125.678} C_DIS
LIN {X 0.246,Y -456.208,Z 643.496,A 0.000,B 0.000,C 90.000,E1 125.231} C_DIS
LIN {X 0.033,Y -463.847,Z 643.493,A 0.000,B 0.000,C 90.000,E1 124.739} C_DIS
LIN {X 0.030,Y -473.344,Z 643.489,A 0.000,B 0.000,C 90.000,E1 124.072} C_DIS
LIN {X -0.047,Y -479.506,Z 643.487,A 0.000,B 0.000,C 90.000,E1 123.627} C_DIS
LIN {X -0.254,Y -488.590,Z 643.483,A 0.000,B 0.000,C 90.000,E1 122.959} C_DIS
LIN {X -0.115,Y -494.484,Z 643.480,A 0.000,B 0.000,C 90.000,E1 122.467} C_DIS
LIN {X -0.158,Y -500.035,Z 643.478,A 0.000,B 0.000,C 90.000,E1 122.005} C_DIS
LIN {X -0.229,Y -508.806,Z 643.474,A 0.000,B 0.000,C 90.000,E1 121.258} C_DIS
LIN {X 0.158,Y -517.073,Z 643.469,A 0.000,B 0.000,C 90.000,E1 120.463} C_DIS
LIN {X 0.266,Y -523.905,Z 643.466,A 0.000,B 0.000,C 90.000,E1 119.795} C_DIS
LIN {X 0.030,Y -529.246,Z 643.463,A 0.000,B 0.000,C 90.000,E1 119.283} C_DIS
LIN {X 0.013,Y -533.262,Z 643.460,A 0.000,B 0.000,C 90.000,E1 118.871} C_DIS
LIN {X -0.271,Y -538.074,Z 643.457,A 0.000,B 0.000,C 90.000,E1 118.359} C_DIS
LIN {X -0.070,Y -542.704,Z 643.454,A 0.000,B 0.000,C 90.000,E1 117.769} C_DIS
LIN {X -0.104,Y -546.817,Z 643.451,A 0.000,B 0.000,C 90.000,E1 117.206} C_DIS
LIN {X 0.025,Y -551.273,Z 643.447,A 0.000,B 0.000,C 90.000,E1 116.488} C_DIS
LIN {X 0.080,Y -555.799,Z 643.443,A 0.000,B 0.000,C 90.000,E1 115.668} C_DIS
LIN {X 0.046,Y -559.304,Z 643.439,A 0.000,B 0.000,C 90.000,E1 114.975} C_DIS
LIN {X 0.046,Y -562.495,Z 643.435,A 0.000,B 0.000,C 90.000,E1 114.283} C_DIS
LIN {X -0.025,Y -566.007,Z 643.430,A 0.000,B 0.000,C 90.000,E1 113.462} C_DIS
LIN {X 0.277,Y -570.381,Z 643.424,A 0.000,B 0.000,C 90.000,E1 112.333} C_DIS
LIN {X -0.114,Y -574.172,Z 643.418,A 0.000,B 0.000,C 90.000,E1 111.280} C_DIS
LIN {X 0.079,Y -577.484,Z 643.412,A 0.000,B 0.000,C 90.000,E1 110.174} C_DIS
LIN {X -0.264,Y -579.762,Z 643.408,A 0.000,B 0.000,C 90.000,E1 109.396} C_DIS
LIN {X -0.184,Y -582.420,Z 643.402,A 0.000,B 0.000,C 90.000,E1 108.308} C_DIS
LIN {X 0.269,Y -584.239,Z 643.397,A 0.000,B 0.000,C 90.000,E1 107.457} C_DIS
LIN {X -0.321,Y -589.013,Z 643.385,A 0.000,B 0.000,C 90.000,E1 105.371} C_DIS
LIN {X -0.021,Y -592.124,Z 643.378,A 0.000,B 0.000,C 90.000,E1 104.008} C_DIS
LIN {X 0.330,Y -595.274,Z 643.370,A 0.000,B 0.000,C 90.000,E1 102.647} C_DIS
LIN {X -0.105,Y -598.292,Z 643.363,A 0.000,B 0.000,C 90.000,E1 101.366} C_DIS
LIN {X 0.214,Y -601.259,Z 643.356,A 0.000,B 0.000,C 90.000,E1 100.018} C_DIS
LIN {X -0.218,Y -604.148,Z 643.349,A 0.000,B 0.000,C 90.000,E1 98.746} C_DIS
LIN {X -0.233,Y -606.314,Z 643.343,A 0.000,B 0.000,C 90.000,E1 97.701} C_DIS
LIN {X 0.021,Y -608.790,Z 643.335,A 0.000,B 0.000,C 90.000,E1 96.372} C_DIS
LIN {X 0.254,Y -610.967,Z 643.328,A 0.000,B 0.000,C 90.000,E1 95.049} C_DIS
LIN {X 0.242,Y -612.622,Z 643.322,A 0.000,B 0.000,C 90.000,E1 94.012} C_DIS
LIN {X -0.117,Y -614.439,Z 643.315,A 0.000,B 0.000,C 90.000,E1 92.751} C_DIS
LIN {X -0.132,Y -615.663,Z 643.310,A 0.000,B 0.000,C 90.000,E1 91.718} C_DIS
LIN {X 0.162,Y -616.399,Z 643.305,A 0.000,B 0.000,C 90.000,E1 90.917} C_DIS
LIN {X -0.148,Y -617.395,Z 643.298,A 0.000,B 0.000,C 90.000,E1 89.656} C_DIS
LIN {X 0.172,Y -618.011,Z 643.291,A 0.000,B 0.000,C 90.000,E1 88.339} C_DIS
LIN {X -0.108,Y -618.220,Z 643.287,A 0.000,B 0.000,C 90.000,E1 87.593} C_DIS
LIN {X 0.242,Y -618.212,Z 643.279,A 0.000,B 0.000,C 90.000,E1 86.274} C_DIS
LIN {X 0.275,Y -618.003,Z 643.274,A 0.000,B 0.000,C 90.000,E1 85.241} C_DIS
LIN {X -0.257,Y -617.552,Z 643.268,A 0.000,B 0.000,C 90.000,E1 84.261} C_DIS
LIN {X 0.186,Y -616.765,Z 643.261,A 0.000,B 0.000,C 90.000,E1 82.932} C_DIS
LIN {X 0.255,Y -615.995,Z 643.255,A 0.000,B 0.000,C 90.000,E1 81.894} C_DIS
LIN {X -0.210,Y -614.838,Z 643.249,A 0.000,B 0.000,C 90.000,E1 80.905} C_DIS
LIN {X 0.168,Y -613.169,Z 643.242,A 0.000,B 0.000,C 90.000,E1 79.577} C_DIS
LIN {X 0.131,Y -611.181,Z 643.235,A 0.000,B 0.000,C 90.000,E1 78.285} C_DIS
LIN {X 0.073,Y -609.021,Z 643.228,A 0.000,B 0.000,C 90.000,E1 76.992} C_DIS
LIN {X 0.234,Y -607.155,Z 643.222,A 0.000,B 0.000,C 90.000,E1 75.936} C_DIS
LIN {X 0.252,Y -604.676,Z 643.215,A 0.000,B 0.000,C 90.000,E1 74.629} C_DIS
LIN {X 0.224,Y -601.899,Z 643.208,A 0.000,B 0.000,C 90.000,E1 73.323} C_DIS
LIN {X 0.318,Y -598.996,Z 643.200,A 0.000,B 0.000,C 90.000,E1 72.000} C_DIS
LIN {X 0.093,Y -596.396,Z 643.194,A 0.000,B 0.000,C 90.000,E1 70.967} C_DIS
LIN {X 0.251,Y -594.960,Z 643.191,A 0.000,B 0.000,C 90.000,E1 70.423} C_DIS
LIN {X -0.161,Y -593.471,Z 643.188,A 0.000,B 0.000,C 90.000,E1 69.934} C_DIS
LIN {X -0.137,Y -591.043,Z 643.184,A 0.000,B 0.000,C 90.000,E1 69.135} C_DIS
LIN {X -0.137,Y -588.369,Z 643.180,A 0.000,B 0.000,C 90.000,E1 68.337} C_DIS
LIN {X 0.251,Y -584.390,Z 643.174,A 0.000,B 0.000,C 90.000,E1 67.230} C_DIS
LIN {X 0.170,Y -581.222,Z 643.169,A 0.000,B 0.000,C 90.000,E1 66.433} C_DIS
LIN {X -0.241,Y -577.800,Z 643.165,A 0.000,B 0.000,C 90.000,E1 65.665} C_DIS
LIN {X -0.229,Y -573.616,Z 643.159,A 0.000,B 0.000,C 90.000,E1 64.717} C_DIS
LIN {X -0.194,Y -569.572,Z 643.155,A 0.000,B 0.000,C 90.000,E1 63.896} C_DIS
LIN {X 0.039,Y -566.082,Z 643.151,A 0.000,B 0.000,C 90.000,E1 63.204} C_DIS
LIN {X -0.165,Y -562.080,Z 643.147,A 0.000,B 0.000,C 90.000,E1 62.538} C_DIS
LIN {X -0.240,Y -558.029,Z 643.144,A 0.000,B 0.000,C 90.000,E1 61.897} C_DIS
LIN {X 0.096,Y -554.181,Z 643.141,A 0.000,B 0.000,C 90.000,E1 61.307} C_DIS
LIN {X -0.348,Y -549.889,Z 643.138,A 0.000,B 0.000,C 90.000,E1 60.795} C_DIS
LIN {X -0.074,Y -545.103,Z 643.134,A 0.000,B 0.000,C 90.000,E1 60.205} C_DIS
LIN {X -0.147,Y -539.731,Z 643.131,A 0.000,B 0.000,C 90.000,E1 59.665} C_DIS
LIN {X -0.047,Y -535.373,Z 643.129,A 0.000,B 0.000,C 90.000,E1 59.253} C_DIS
LIN {X 0.169,Y -529.308,Z 643.126,A 0.000,B 0.000,C 90.000,E1 58.742} C_DIS
LIN {X 0.010,Y -522.108,Z 643.124,A 0.000,B 0.000,C 90.000,E1 58.250} C_DIS
LIN {X -0.288,Y -515.342,Z 643.121,A 0.000,B 0.000,C 90.000,E1 57.867} C_DIS
LIN {X -0.107,Y -507.036,Z 643.119,A 0.000,B 0.000,C 90.000,E1 57.375} C_DIS
LIN {X 0.004,Y -483.842,Z 643.112,A 0.000,B 0.000,C 90.000,E1 56.167} C_DIS
LIN {X 0.099,Y -461.980,Z 643.106,A 0.000,B 0.000,C 90.000,E1 55.022} C_DIS
LIN {X 0.229,Y -441.966,Z 643.100,A 0.000,B 0.000,C 90.000,E1 53.909} C_DIS
LIN {X -0.288,Y -437.195,Z 643.098,A 0.000,B 0.000,C 90.000,E1 53.703} C_DIS
LIN {X 0.022,Y -437.119,Z 643.098,A 0.000,B 0.000,C 90.000,E1 53.657} C_DIS
LIN {X -0.028,Y -431.707,Z 643.083,A 0.000,B 0.000,C 90.000,E1 50.928} C_DIS
LIN {X -0.120,Y -430.100,Z 643.079,A 0.000,B 0.000,C 90.000,E1 50.275} C_DIS
LIN {X 0.060,Y -422.848,Z 643.062,A 0.000,B 0.000,C 90.000,E1 47.067} C_DIS
LIN {X -0.080,Y -423.211,Z 643.053,A 0.000,B 0.000,C 90.000,E1 45.567} C_DIS
LIN {X 0.224,Y -423.321,Z 643.048,A 0.000,B 0.000,C 90.000,E1 44.514} C_DIS
LIN {X 0.056,Y -423.826,Z 643.033,A 0.000,B 0.000,C 90.000,E1 41.838} C_DIS
LIN {X 0.029,Y -424.589,Z 643.019,A 0.000,B 0.000,C 90.000,E1 39.483} C_DIS
LIN {X -0.189,Y -425.644,Z 643.006,A 0.000,B 0.000,C 90.000,E1 37.156} C_DIS
LIN {X 0.077,Y -426.667,Z 642.995,A 0.000,B 0.000,C 90.000,E1 35.105} C_DIS
LIN {X 0.108,Y -427.720,Z 642.982,A 0.000,B 0.000,C 90.000,E1 32.752} C_DIS
LIN {X 0.079,Y -428.538,Z 642.973,A 0.000,B 0.000,C 90.000,E1 31.082} C_DIS
LIN {X 0.063,Y -429.379,Z 642.962,A 0.000,B 0.000,C 90.000,E1 29.077} C_DIS
LIN {X 0.026,Y -430.314,Z 642.951,A 0.000,B 0.000,C 90.000,E1 27.078} C_DIS
LIN {X 0.205,Y -431.014,Z 642.943,A 0.000,B 0.000,C 90.000,E1 25.720} C_DIS
LIN {X 0.217,Y -432.471,Z 642.930,A 0.000,B 0.000,C 90.000,E1 23.387} C_DIS
LIN {X 0.102,Y -433.848,Z 642.919,A 0.000,B 0.000,C 90.000,E1 21.408} C_DIS
LIN {X 0.037,Y -434.920,Z 642.910,A 0.000,B 0.000,C 90.000,E1 19.758} C_DIS
LIN {X 0.161,Y -435.713,Z 642.902,A 0.000,B 0.000,C 90.000,E1 18.417} C_DIS
LIN {X 0.157,Y -436.475,Z 642.895,A 0.000,B 0.000,C 90.000,E1 17.094} C_DIS
LIN {X -0.189,Y -437.977,Z 642.882,A 0.000,B 0.000,C 90.000,E1 14.828} C_DIS
LIN {X -0.148,Y -439.271,Z 642.873,A 0.000,B 0.000,C 90.000,E1 13.175} C_DIS
LIN {X -0.150,Y -441.427,Z 642.859,A 0.000,B 0.000,C 90.000,E1 10.546} C_DIS
LIN {X -0.060,Y -444.291,Z 642.842,A 0.000,B 0.000,C 90.000,E1 7.587} C_DIS
LIN {X -0.023,Y -446.366,Z 642.831,A 0.000,B 0.000,C 90.000,E1 5.625} C_DIS
LIN {X -0.112,Y -449.457,Z 642.817,A 0.000,B 0.000,C 90.000,E1 3.037} C_DIS
LIN {X -0.178,Y -452.880,Z 642.802,A 0.000,B 0.000,C 90.000,E1 0.458} C_DIS
LIN {X -0.117,Y -456.702,Z 642.788,A 0.000,B 0.000,C 90.000,E1 357.879} C_DIS
LIN {X 0.145,Y -459.895,Z 642.778,A 0.000,B 0.000,C 90.000,E1 355.927} C_DIS
LIN {X -0.203,Y -463.735,Z 642.765,A 0.000,B 0.000,C 90.000,E1 353.742} C_DIS
LIN {X -0.162,Y -465.961,Z 642.758,A 0.000,B 0.000,C 90.000,E1 352.470} C_DIS
LIN {X 0.002,Y -469.277,Z 642.748,A 0.000,B 0.000,C 90.000,E1 350.557} C_DIS
LIN {X 0.121,Y -471.456,Z 642.741,A 0.000,B 0.000,C 90.000,E1 349.285} C_DIS
LIN {X -0.055,Y -475.253,Z 642.728,A 0.000,B 0.000,C 90.000,E1 347.117} C_DIS
LIN {X -0.021,Y -479.276,Z 642.716,A 0.000,B 0.000,C 90.000,E1 344.936} C_DIS
LIN {X -0.089,Y -483.367,Z 642.704,A 0.000,B 0.000,C 90.000,E1 342.779} C_DIS
LIN {X 0.096,Y -486.962,Z 642.694,A 0.000,B 0.000,C 90.000,E1 340.913} C_DIS
LIN {X 0.091,Y -491.196,Z 642.682,A 0.000,B 0.000,C 90.000,E1 338.773} C_DIS
LIN {X 0.240,Y -493.506,Z 642.675,A 0.000,B 0.000,C 90.000,E1 337.539} C_DIS
LIN {X 0.015,Y -496.092,Z 642.667,A 0.000,B 0.000,C 90.000,E1 336.049} C_DIS
LIN {X -0.020,Y -498.021,Z 642.660,A 0.000,B 0.000,C 90.000,E1 334.845} C_DIS
LIN {X 0.031,Y -500.470,Z 642.652,A 0.000,B 0.000,C 90.000,E1 333.332} C_DIS
LIN {X 0.122,Y -504.349,Z 642.639,A 0.000,B 0.000,C 90.000,E1 330.923} C_DIS
LIN {X 0.194,Y -507.740,Z 642.629,A 0.000,B 0.000,C 90.000,E1 329.125} C_DIS
LIN {X 0.044,Y -509.988,Z 642.624,A 0.000,B 0.000,C 90.000,E1 328.250} C_DIS
LIN {X 0.107,Y -510.808,Z 642.622,A 0.000,B 0.000,C 90.000,E1 327.946} C_DIS
LIN {X -0.175,Y -512.350,Z 642.620,A 0.000,B 0.000,C 90.000,E1 327.533} C_DIS
LIN {X 0.110,Y -514.703,Z 642.617,A 0.000,B 0.000,C 90.000,E1 326.993} C_DIS
LIN {X -0.127,Y -517.863,Z 642.614,A 0.000,B 0.000,C 90.000,E1 326.548} C_DIS
LIN {X -0.215,Y -520.669,Z 642.612,A 0.000,B 0.000,C 90.000,E1 326.215} C_DIS
LIN {X -0.313,Y -526.502,Z 642.609,A 0.000,B 0.000,C 90.000,E1 325.674} C_DIS
LIN {X 0.274,Y -544.880,Z 642.601,A 0.000,B 0.000,C 90.000,E1 324.116} C_DIS
LIN {X -0.191,Y -554.900,Z 642.596,A 0.000,B 0.000,C 90.000,E1 323.336} C_DIS
LIN {X -0.047,Y -566.073,Z 642.591,A 0.000,B 0.000,C 90.000,E1 322.351} C_DIS
LIN {X -0.109,Y -578.315,Z 642.585,A 0.000,B 0.000,C 90.000,E1 321.251} C_DIS
LIN {X 0.229,Y -587.710,Z 642.580,A 0.000,B 0.000,C 90.000,E1 320.356} C_DIS
LIN {X 0.147,Y -594.324,Z 642.576,A 0.000,B 0.000,C 90.000,E1 319.747} C_DIS
LIN {X 0.213,Y -601.844,Z 642.572,A 0.000,B 0.000,C 90.000,E1 319.013} C_DIS
LIN {X 0.054,Y -606.776,Z 642.570,A 0.000,B 0.000,C 90.000,E1 318.528} C_DIS
LIN {X 0.205,Y -611.365,Z 642.567,A 0.000,B 0.000,C 90.000,E1 318.000} C_DIS
LIN {X 0.293,Y -616.644,Z 642.563,A 0.000,B 0.000,C 90.000,E1 317.391} C_DIS
LIN {X -0.088,Y -621.906,Z 642.560,A 0.000,B 0.000,C 90.000,E1 316.782} C_DIS
LIN {X -0.004,Y -626.754,Z 642.556,A 0.000,B 0.000,C 90.000,E1 316.134} C_DIS
LIN {X 0.127,Y -631.416,Z 642.553,A 0.000,B 0.000,C 90.000,E1 315.486} C_DIS
LIN {X 0.270,Y -637.626,Z 642.548,A 0.000,B 0.000,C 90.000,E1 314.595} C_DIS
LIN {X -0.079,Y -644.441,Z 642.542,A 0.000,B 0.000,C 90.000,E1 313.623} C_DIS
LIN {X -0.278,Y -650.246,Z 642.538,A 0.000,B 0.000,C 90.000,E1 312.771} C_DIS
LIN {X 0.047,Y -654.940,Z 642.533,A 0.000,B 0.000,C 90.000,E1 312.000} C_DIS
LIN {X -0.072,Y -659.481,Z 642.529,A 0.000,B 0.000,C 90.000,E1 311.272} C_DIS
LIN {X -0.091,Y -663.461,Z 642.525,A 0.000,B 0.000,C 90.000,E1 310.539} C_DIS
LIN {X 0.401,Y -667.764,Z 642.521,A 0.000,B 0.000,C 90.000,E1 309.644} C_DIS
LIN {X -0.050,Y -671.112,Z 642.516,A 0.000,B 0.000,C 90.000,E1 308.955} C_DIS
LIN {X 0.046,Y -673.197,Z 642.514,A 0.000,B 0.000,C 90.000,E1 308.463} C_DIS
LIN {X -0.244,Y -676.891,Z 642.508,A 0.000,B 0.000,C 90.000,E1 307.523} C_DIS
LIN {X -0.100,Y -678.626,Z 642.506,A 0.000,B 0.000,C 90.000,E1 307.030} C_DIS
LIN {X -0.320,Y -681.806,Z 642.500,A 0.000,B 0.000,C 90.000,E1 306.091} C_DIS
LIN {X 0.048,Y -684.771,Z 642.495,A 0.000,B 0.000,C 90.000,E1 305.105} C_DIS
LIN {X 0.083,Y -688.307,Z 642.488,A 0.000,B 0.000,C 90.000,E1 303.913} C_DIS
LIN {X 0.149,Y -690.891,Z 642.483,A 0.000,B 0.000,C 90.000,E1 302.959} C_DIS
LIN {X 0.250,Y -693.316,Z 642.478,A 0.000,B 0.000,C 90.000,E1 302.005} C_DIS
LIN {X 0.025,Y -696.103,Z 642.471,A 0.000,B 0.000,C 90.000,E1 300.846} C_DIS
LIN {X -0.175,Y -698.243,Z 642.466,A 0.000,B 0.000,C 90.000,E1 299.922} C_DIS
LIN {X 0.263,Y -700.162,Z 642.461,A 0.000,B 0.000,C 90.000,E1 298.949} C_DIS
LIN {X 0.114,Y -701.898,Z 642.456,A 0.000,B 0.000,C 90.000,E1 298.025} C_DIS
LIN {X -0.344,Y -703.421,Z 642.451,A 0.000,B 0.000,C 90.000,E1 297.129} C_DIS
LIN {X -0.124,Y -704.303,Z 642.447,A 0.000,B 0.000,C 90.000,E1 296.411} C_DIS
LIN {X 0.160,Y -704.530,Z 642.445,A 0.000,B 0.000,C 90.000,E1 296.155} C_DIS
LIN {X -0.209,Y -704.707,Z 642.443,A 0.000,B 0.000,C 90.000,E1 295.720} C_DIS
LIN {X 0.078,Y -704.550,Z 642.442,A 0.000,B 0.000,C 90.000,E1 295.463} C_DIS
LIN {X -0.285,Y -703.580,Z 642.439,A 0.000,B 0.000,C 90.000,E1 295.027} C_DIS
LIN {X -0.001,Y -702.657,Z 642.438,A 0.000,B 0.000,C 90.000,E1 294.771} C_DIS
LIN {X -0.371,Y -699.447,Z 642.435,A 0.000,B 0.000,C 90.000,E1 294.335} C_DIS
LIN {X -0.237,Y -698.455,Z 642.434,A 0.000,B 0.000,C 90.000,E1 294.207} C_DIS
LIN {X -0.102,Y -696.965,Z 642.434,A 0.000,B 0.000,C 90.000,E1 294.079} C_DIS
LIN {X 0.181,Y -694.846,Z 642.433,A 0.000,B 0.000,C 90.000,E1 293.951} C_DIS
LIN {X 0.261,Y -690.555,Z 642.432,A 0.000,B 0.000,C 90.000,E1 293.770} C_DIS
LIN {X 0.317,Y -686.710,Z 642.432,A 0.000,B 0.000,C 90.000,E1 293.643} C_DIS
LIN {X 0.232,Y -680.681,Z 642.431,A 0.000,B 0.000,C 90.000,E1 293.515} C_DIS
LIN {X -0.069,Y -672.190,Z 642.430,A 0.000,B 0.000,C 90.000,E1 293.439} C_DIS
LIN {X -0.156,Y -665.588,Z 642.430,A 0.000,B 0.000,C 90.000,E1 293.387} C_DIS
LIN {X -0.132,Y -652.519,Z 642.429,A 0.000,B 0.000,C 90.000,E1 293.206} C_DIS
LIN {X 0.021,Y -642.706,Z 642.428,A 0.000,B 0.000,C 90.000,E1 293.025} C_DIS
LIN {X 0.079,Y -633.094,Z 642.427,A 0.000,B 0.000,C 90.000,E1 292.823} C_DIS
LIN {X -0.004,Y -623.123,Z 642.426,A 0.000,B 0.000,C 90.000,E1 292.589} C_DIS
LIN {X 0.096,Y -609.830,Z 642.423,A 0.000,B 0.000,C 90.000,E1 292.206} C_DIS
LIN {X 0.003,Y -582.089,Z 642.419,A 0.000,B 0.000,C 90.000,E1 291.354} C_DIS
LIN {X -0.161,Y -574.932,Z 642.417,A 0.000,B 0.000,C 90.000,E1 291.153} C_DIS
LIN {X -0.146,Y -564.528,Z 642.416,A 0.000,B 0.000,C 90.000,E1 290.844} C_DIS
LIN {X 0.151,Y -559.642,Z 642.415,A 0.000,B 0.000,C 90.000,E1 290.610} C_DIS
LIN {X 0.007,Y -556.745,Z 642.414,A 0.000,B 0.000,C 90.000,E1 290.429} C_DIS
LIN {X -0.045,Y -556.680,Z 642.414,A 0.000,B 0.000,C 90.000,E1 290.429} C_DIS
LIN {X 0.054,Y -555.995,Z 642.413,A 0.000,B 0.000,C 90.000,E1 290.248} C_DIS
LIN {X 0.229,Y -555.534,Z 642.410,A 0.000,B 0.000,C 90.000,E1 289.812} C_DIS
LIN {X 0.254,Y -555.444,Z 642.403,A 0.000,B 0.000,C 90.000,E1 288.417} C_DIS
LIN {X 0.100,Y -555.200,Z 642.395,A 0.000,B 0.000,C 90.000,E1 287.040} C_DIS
LIN {X -0.176,Y -554.899,Z 642.389,A 0.000,B 0.000,C 90.000,E1 285.953} C_DIS
LIN {X 0.040,Y -554.318,Z 642.381,A 0.000,B 0.000,C 90.000,E1 284.537} C_DIS
LIN {X 0.252,Y -553.600,Z 642.373,A 0.000,B 0.000,C 90.000,E1 283.119} C_DIS
LIN {X 0.151,Y -552.472,Z 642.361,A 0.000,B 0.000,C 90.000,E1 280.894} C_DIS
LIN {X -0.093,Y -551.605,Z 642.348,A 0.000,B 0.000,C 90.000,E1 278.681} C_DIS
LIN {X 0.012,Y -550.793,Z 642.336,A 0.000,B 0.000,C 90.000,E1 276.429} C_DIS
LIN {X -0.059,Y -550.288,Z 642.325,A 0.000,B 0.000,C 90.000,E1 274.473} C_DIS
LIN {X 0.266,Y -549.968,Z 642.317,A 0.000,B 0.000,C 90.000,E1 273.037} C_DIS
LIN {X 0.000,Y -549.576,Z 642.309,A 0.000,B 0.000,C 90.000,E1 271.661} C_DIS
LIN {X -0.230,Y -548.977,Z 642.300,A 0.000,B 0.000,C 90.000,E1 270.000} C_DIS
LIN {X 0.026,Y -548.228,Z 642.292,A 0.000,B 0.000,C 90.000,E1 268.568} C_DIS
LIN {X -0.225,Y -547.468,Z 642.283,A 0.000,B 0.000,C 90.000,E1 266.906} C_DIS
LIN {X 0.009,Y -546.880,Z 642.276,A 0.000,B 0.000,C 90.000,E1 265.755} C_DIS
LIN {X 0.192,Y -546.053,Z 642.270,A 0.000,B 0.000,C 90.000,E1 264.609} C_DIS
LIN {X -0.052,Y -545.006,Z 642.262,A 0.000,B 0.000,C 90.000,E1 263.223} C_DIS
LIN {X 0.135,Y -544.235,Z 642.258,A 0.000,B 0.000,C 90.000,E1 262.356} C_DIS
LIN {X -0.143,Y -542.655,Z 642.250,A 0.000,B 0.000,C 90.000,E1 260.971} C_DIS
LIN {X -0.067,Y -540.153,Z 642.236,A 0.000,B 0.000,C 90.000,E1 258.409} C_DIS
LIN {X 0.083,Y -538.220,Z 642.223,A 0.000,B 0.000,C 90.000,E1 256.117} C_DIS
LIN {X -0.059,Y -537.274,Z 642.217,A 0.000,B 0.000,C 90.000,E1 254.991} C_DIS
LIN {X -0.016,Y -535.902,Z 642.209,A 0.000,B 0.000,C 90.000,E1 253.559} C_DIS
LIN {X -0.076,Y -533.730,Z 642.196,A 0.000,B 0.000,C 90.000,E1 251.275} C_DIS
LIN {X -0.156,Y -532.837,Z 642.191,A 0.000,B 0.000,C 90.000,E1 250.423} C_DIS
LIN {X -0.050,Y -531.286,Z 642.185,A 0.000,B 0.000,C 90.000,E1 249.263} C_DIS
LIN {X 0.216,Y -529.230,Z 642.177,A 0.000,B 0.000,C 90.000,E1 247.794} C_DIS
LIN {X 0.278,Y -527.868,Z 642.172,A 0.000,B 0.000,C 90.000,E1 246.922} C_DIS
LIN {X 0.018,Y -525.939,Z 642.166,A 0.000,B 0.000,C 90.000,E1 245.793} C_DIS
LIN {X -0.271,Y -523.695,Z 642.159,A 0.000,B 0.000,C 90.000,E1 244.665} C_DIS
LIN {X -0.049,Y -521.911,Z 642.154,A 0.000,B 0.000,C 90.000,E1 243.768} C_DIS
LIN {X -0.125,Y -518.227,Z 642.145,A 0.000,B 0.000,C 90.000,E1 242.025} C_DIS
LIN {X 0.053,Y -515.115,Z 642.136,A 0.000,B 0.000,C 90.000,E1 240.539} C_DIS
LIN {X 0.327,Y -512.393,Z 642.130,A 0.000,B 0.000,C 90.000,E1 239.331} C_DIS
LIN {X 0.099,Y -508.200,Z 642.120,A 0.000,B 0.000,C 90.000,E1 237.582} C_DIS
LIN {X 0.159,Y -504.678,Z 642.112,A 0.000,B 0.000,C 90.000,E1 236.087} C_DIS
LIN {X 0.018,Y -500.853,Z 642.103,A 0.000,B 0.000,C 90.000,E1 234.609} C_DIS
LIN {X 0.075,Y -496.115,Z 642.093,A 0.000,B 0.000,C 90.000,E1 232.798} C_DIS
LIN {X 0.066,Y -490.885,Z 642.082,A 0.000,B 0.000,C 90.000,E1 230.678} C_DIS
LIN {X 0.036,Y -486.451,Z 642.071,A 0.000,B 0.000,C 90.000,E1 228.852} C_DIS
LIN {X 0.038,Y -481.330,Z 642.060,A 0.000,B 0.000,C 90.000,E1 226.701} C_DIS
LIN {X -0.135,Y -478.338,Z 642.053,A 0.000,B 0.000,C 90.000,E1 225.486} C_DIS
LIN {X -0.239,Y -474.617,Z 642.044,A 0.000,B 0.000,C 90.000,E1 223.947} C_DIS
LIN {X -0.077,Y -471.035,Z 642.035,A 0.000,B 0.000,C 90.000,E1 222.366} C_DIS
LIN {X -0.059,Y -465.547,Z 642.021,A 0.000,B 0.000,C 90.000,E1 219.850} C_DIS
LIN {X 0.061,Y -461.495,Z 642.011,A 0.000,B 0.000,C 90.000,E1 217.935} C_DIS
LIN {X 0.012,Y -456.357,Z 641.997,A 0.000,B 0.000,C 90.000,E1 215.391} C_DIS
LIN {X 0.027,Y -453.462,Z 641.988,A 0.000,B 0.000,C 90.000,E1 213.785} C_DIS
LIN {X 0.065,Y -448.186,Z 641.972,A 0.000,B 0.000,C 90.000,E1 210.875} C_DIS
LIN {X -0.114,Y -444.765,Z 641.961,A 0.000,B 0.000,C 90.000,E1 208.949} C_DIS
LIN {X -0.204,Y -441.213,Z 641.950,A 0.000,B 0.000,C 90.000,E1 207.001} C_DIS
LIN {X -0.049,Y -438.852,Z 641.943,A 0.000,B 0.000,C 90.000,E1 205.668} C_DIS
LIN {X -0.088,Y -435.193,Z 641.932,A 0.000,B 0.000,C 90.000,E1 203.695} C_DIS
LIN {X 0.011,Y -432.286,Z 641.922,A 0.000,B 0.000,C 90.000,E1 202.025} C_DIS
LIN {X 0.261,Y -428.805,Z 641.911,A 0.000,B 0.000,C 90.000,E1 199.993} C_DIS
LIN {X 0.136,Y -425.445,Z 641.900,A 0.000,B 0.000,C 90.000,E1 198.000} C_DIS
LIN {X -0.010,Y -421.671,Z 641.887,A 0.000,B 0.000,C 90.000,E1 195.662} C_DIS
LIN {X 0.110,Y -418.982,Z 641.878,A 0.000,B 0.000,C 90.000,E1 193.953} C_DIS
LIN {X -0.173,Y -415.808,Z 641.866,A 0.000,B 0.000,C 90.000,E1 191.951} C_DIS
LIN {X -0.213,Y -412.750,Z 641.855,A 0.000,B 0.000,C 90.000,E1 189.905} C_DIS
LIN {X -0.062,Y -410.794,Z 641.847,A 0.000,B 0.000,C 90.000,E1 188.511} C_DIS
LIN {X 0.010,Y -407.293,Z 641.834,A 0.000,B 0.000,C 90.000,E1 186.087} C_DIS
LIN {X -0.101,Y -403.376,Z 641.817,A 0.000,B 0.000,C 90.000,E1 182.980} C_DIS
LIN {X -0.036,Y -400.014,Z 641.799,A 0.000,B 0.000,C 90.000,E1 179.828} C_DIS
LIN {X 0.029,Y -398.068,Z 641.785,A 0.000,B 0.000,C 90.000,E1 177.364} C_DIS
LIN {X -0.024,Y -396.315,Z 641.768,A 0.000,B 0.000,C 90.000,E1 174.204} C_DIS
LIN {X 0.051,Y -395.555,Z 641.754,A 0.000,B 0.000,C 90.000,E1 171.724} C_DIS
LIN {X -0.103,Y -395.101,Z 641.740,A 0.000,B 0.000,C 90.000,E1 169.275} C_DIS
LIN {X 0.128,Y -394.962,Z 641.723,A 0.000,B 0.000,C 90.000,E1 166.061} C_DIS
LIN {X -0.127,Y -395.057,Z 641.715,A 0.000,B 0.000,C 90.000,E1 164.685} C_DIS
LIN {X 0.021,Y -395.335,Z 641.703,A 0.000,B 0.000,C 90.000,E1 162.543} C_DIS
LIN {X 0.032,Y -395.765,Z 641.691,A 0.000,B 0.000,C 90.000,E1 160.423} C_DIS
LIN {X 0.188,Y -396.187,Z 641.680,A 0.000,B 0.000,C 90.000,E1 158.284} C_DIS
LIN {X 0.127,Y -396.786,Z 641.668,A 0.000,B 0.000,C 90.000,E1 156.177} C_DIS
LIN {X 0.042,Y -397.286,Z 641.656,A 0.000,B 0.000,C 90.000,E1 154.076} C_DIS
LIN {X -0.155,Y -397.919,Z 641.642,A 0.000,B 0.000,C 90.000,E1 151.641} C_DIS
LIN {X -0.074,Y -398.447,Z 641.633,A 0.000,B 0.000,C 90.000,E1 149.871} C_DIS
LIN {X 0.190,Y -399.151,Z 641.619,A 0.000,B 0.000,C 90.000,E1 147.375} C_DIS
LIN {X -0.198,Y -400.054,Z 641.605,A 0.000,B 0.000,C 90.000,E1 144.975} C_DIS
LIN {X 0.011,Y -400.949,Z 641.594,A 0.000,B 0.000,C 90.000,E1 142.844} C_DIS
LIN {X 0.048,Y -401.680,Z 641.584,A 0.000,B 0.000,C 90.000,E1 141.090} C_DIS
LIN {X -0.031,Y -402.281,Z 641.576,A 0.000,B 0.000,C 90.000,E1 139.703} C_DIS
LIN {X -0.026,Y -402.959,Z 641.566,A 0.000,B 0.000,C 90.000,E1 137.957} C_DIS
LIN {X -0.207,Y -403.772,Z 641.555,A 0.000,B 0.000,C 90.000,E1 135.891} C_DIS
LIN {X 0.047,Y -404.881,Z 641.541,A 0.000,B 0.000,C 90.000,E1 133.419} C_DIS
LIN {X 0.051,Y -406.319,Z 641.528,A 0.000,B 0.000,C 90.000,E1 130.987} C_DIS
LIN {X 0.165,Y -407.451,Z 641.522,A 0.000,B 0.000,C 90.000,E1 129.930} C_DIS
LIN {X -0.163,Y -408.978,Z 641.517,A 0.000,B 0.000,C 90.000,E1 129.116} C_DIS
LIN {X -0.094,Y -410.671,Z 641.514,A 0.000,B 0.000,C 90.000,E1 128.588} C_DIS
LIN {X 0.186,Y -410.894,Z 641.514,A 0.000,B 0.000,C 90.000,E1 128.463} C_DIS
LIN {X 0.053,Y -413.465,Z 641.511,A 0.000,B 0.000,C 90.000,E1 128.051} C_DIS
LIN {X -0.027,Y -414.923,Z 641.511,A 0.000,B 0.000,C 90.000,E1 127.890} C_DIS
LIN {X 0.027,Y -416.388,Z 641.510,A 0.000,B 0.000,C 90.000,E1 127.729} C_DIS
LIN {X -0.081,Y -422.190,Z 641.507,A 0.000,B 0.000,C 90.000,E1 127.282} C_DIS
LIN {X -0.037,Y -450.621,Z 641.497,A 0.000,B 0.000,C 90.000,E1 125.438} C_DIS
LIN {X -0.151,Y -460.439,Z 641.493,A 0.000,B 0.000,C 90.000,E1 124.818} C_DIS
LIN {X 0.075,Y -473.028,Z 641.489,A 0.000,B 0.000,C 90.000,E1 123.913} C_DIS
LIN {X -0.181,Y -480.823,Z 641.485,A 0.000,B 0.000,C 90.000,E1 123.372} C_DIS
LIN {X 0.133,Y -488.522,Z 641.482,A 0.000,B 0.000,C 90.000,E1 122.752} C_DIS
LIN {X -0.006,Y -494.524,Z 641.479,A 0.000,B 0.000,C 90.000,E1 122.291} C_DIS
LIN {X 0.277,Y -500.069,Z 641.477,A 0.000,B 0.000,C 90.000,E1 121.799} C_DIS
LIN {X -0.019,Y -508.865,Z 641.473,A 0.000,B 0.000,C 90.000,E1 121.082} C_DIS
LIN {X -0.183,Y -514.538,Z 641.470,A 0.000,B 0.000,C 90.000,E1 120.590} C_DIS
LIN {X -0.084,Y -522.929,Z 641.466,A 0.000,B 0.000,C 90.000,E1 119.795} C_DIS
LIN {X -0.045,Y -529.577,Z 641.462,A 0.000,B 0.000,C 90.000,E1 119.127} C_DIS
LIN {X -0.184,Y -532.295,Z 641.460,A 0.000,B 0.000,C 90.000,E1 118.871} C_DIS
LIN {X 0.091,Y -537.395,Z 641.457,A 0.000,B 0.000,C 90.000,E1 118.281} C_DIS
LIN {X 0.197,Y -542.938,Z 641.453,A 0.000,B 0.000,C 90.000,E1 117.590} C_DIS
LIN {X 0.121,Y -546.852,Z 641.451,A 0.000,B 0.000,C 90.000,E1 117.078} C_DIS
LIN {X -0.003,Y -549.544,Z 641.448,A 0.000,B 0.000,C 90.000,E1 116.668} C_DIS
LIN {X 0.250,Y -551.376,Z 641.447,A 0.000,B 0.000,C 90.000,E1 116.360} C_DIS
LIN {X -0.212,Y -554.684,Z 641.444,A 0.000,B 0.000,C 90.000,E1 115.848} C_DIS
LIN {X 0.141,Y -559.031,Z 641.439,A 0.000,B 0.000,C 90.000,E1 114.975} C_DIS
LIN {X 0.039,Y -562.891,Z 641.434,A 0.000,B 0.000,C 90.000,E1 114.155} C_DIS
LIN {X 0.069,Y -565.919,Z 641.430,A 0.000,B 0.000,C 90.000,E1 113.462} C_DIS
LIN {X -0.156,Y -570.348,Z 641.424,A 0.000,B 0.000,C 90.000,E1 112.386} C_DIS
LIN {X 0.155,Y -573.278,Z 641.420,A 0.000,B 0.000,C 90.000,E1 111.535} C_DIS
LIN {X -0.030,Y -575.975,Z 641.415,A 0.000,B 0.000,C 90.000,E1 110.737} C_DIS
LIN {X -0.189,Y -578.387,Z 641.411,A 0.000,B 0.000,C 90.000,E1 109.939} C_DIS
LIN {X 0.220,Y -580.622,Z 641.406,A 0.000,B 0.000,C 90.000,E1 109.087} C_DIS
LIN {X -0.082,Y -582.664,Z 641.402,A 0.000,B 0.000,C 90.000,E1 108.308} C_DIS
LIN {X 0.040,Y -585.087,Z 641.396,A 0.000,B 0.000,C 90.000,E1 107.221} C_DIS
LIN {X -0.117,Y -590.588,Z 641.382,A 0.000,B 0.000,C 90.000,E1 104.828} C_DIS
LIN {X 0.176,Y -594.996,Z 641.372,A 0.000,B 0.000,C 90.000,E1 102.939} C_DIS
LIN {X -0.269,Y -598.080,Z 641.365,A 0.000,B 0.000,C 90.000,E1 101.658} C_DIS
LIN {X -0.238,Y -601.742,Z 641.356,A 0.000,B 0.000,C 90.000,E1 100.074} C_DIS
LIN {X -0.068,Y -604.658,Z 641.349,A 0.000,B 0.000,C 90.000,E1 98.746} C_DIS
LIN {X -0.077,Y -606.870,Z 641.343,A 0.000,B 0.000,C 90.000,E1 97.701} C_DIS
LIN {X 0.189,Y -609.375,Z 641.336,A 0.000,B 0.000,C 90.000,E1 96.372} C_DIS
LIN {X -0.177,Y -611.617,Z 641.328,A 0.000,B 0.000,C 90.000,E1 95.106} C_DIS
LIN {X -0.226,Y -613.246,Z 641.323,A 0.000,B 0.000,C 90.000,E1 94.073} C_DIS
LIN {X -0.213,Y -614.758,Z 641.317,A 0.000,B 0.000,C 90.000,E1 93.037} C_DIS
LIN {X 0.065,Y -615.748,Z 641.313,A 0.000,B 0.000,C 90.000,E1 92.236} C_DIS
LIN {X 0.069,Y -616.886,Z 641.307,A 0.000,B 0.000,C 90.000,E1 91.203} C_DIS
LIN {X -0.234,Y -617.912,Z 641.300,A 0.000,B 0.000,C 90.000,E1 89.943} C_DIS
LIN {X -0.217,Y -618.536,Z 641.294,A 0.000,B 0.000,C 90.000,E1 88.912} C_DIS
LIN {X -0.177,Y -618.903,Z 641.288,A 0.000,B 0.000,C 90.000,E1 87.879} C_DIS
LIN {X 0.148,Y -618.969,Z 641.284,A 0.000,B 0.000,C 90.000,E1 87.078} C_DIS
LIN {X 0.193,Y -618.889,Z 641.278,A 0.000,B 0.000,C 90.000,E1 86.045} C_DIS
LIN {X 0.286,Y -618.594,Z 641.272,A 0.000,B 0.000,C 90.000,E1 85.008} C_DIS
LIN {X 0.065,Y -617.928,Z 641.265,A 0.000,B 0.000,C 90.000,E1 83.742} C_DIS
LIN {X 0.150,Y -617.260,Z 641.260,A 0.000,B 0.000,C 90.000,E1 82.704} C_DIS
LIN {X -0.060,Y -616.636,Z 641.255,A 0.000,B 0.000,C 90.000,E1 81.951} C_DIS
LIN {X 0.094,Y -615.445,Z 641.250,A 0.000,B 0.000,C 90.000,E1 80.905} C_DIS
LIN {X -0.120,Y -613.755,Z 641.242,A 0.000,B 0.000,C 90.000,E1 79.634} C_DIS
LIN {X 0.207,Y -611.303,Z 641.234,A 0.000,B 0.000,C 90.000,E1 78.049} C_DIS
LIN {X 0.153,Y -609.069,Z 641.227,A 0.000,B 0.000,C 90.000,E1 76.756} C_DIS
LIN {X 0.314,Y -607.136,Z 641.221,A 0.000,B 0.000,C 90.000,E1 75.700} C_DIS
LIN {X 0.329,Y -604.563,Z 641.214,A 0.000,B 0.000,C 90.000,E1 74.393} C_DIS
LIN {X -0.280,Y -601.689,Z 641.206,A 0.000,B 0.000,C 90.000,E1 73.142} C_DIS
LIN {X 0.102,Y -599.347,Z 641.200,A 0.000,B 0.000,C 90.000,E1 72.054} C_DIS
LIN {X 0.152,Y -596.006,Z 641.193,A 0.000,B 0.000,C 90.000,E1 70.732} C_DIS
LIN {X -0.114,Y -592.868,Z 641.187,A 0.000,B 0.000,C 90.000,E1 69.699} C_DIS
LIN {X -0.099,Y -590.294,Z 641.183,A 0.000,B 0.000,C 90.000,E1 68.901} C_DIS
LIN {X 0.006,Y -588.468,Z 641.180,A 0.000,B 0.000,C 90.000,E1 68.358} C_DIS
LIN {X 0.070,Y -584.393,Z 641.174,A 0.000,B 0.000,C 90.000,E1 67.283} C_DIS
LIN {X -0.005,Y -581.179,Z 641.169,A 0.000,B 0.000,C 90.000,E1 66.485} C_DIS
LIN {X 0.114,Y -577.679,Z 641.165,A 0.000,B 0.000,C 90.000,E1 65.665} C_DIS
LIN {X 0.121,Y -573.437,Z 641.160,A 0.000,B 0.000,C 90.000,E1 64.717} C_DIS
LIN {X 0.153,Y -569.326,Z 641.155,A 0.000,B 0.000,C 90.000,E1 63.896} C_DIS
LIN {X -0.280,Y -565.607,Z 641.151,A 0.000,B 0.000,C 90.000,E1 63.256} C_DIS
LIN {X 0.111,Y -562.393,Z 641.148,A 0.000,B 0.000,C 90.000,E1 62.666} C_DIS
LIN {X 0.070,Y -558.262,Z 641.145,A 0.000,B 0.000,C 90.000,E1 62.025} C_DIS
LIN {X 0.299,Y -553.317,Z 641.141,A 0.000,B 0.000,C 90.000,E1 61.307} C_DIS
LIN {X 0.077,Y -551.003,Z 641.139,A 0.000,B 0.000,C 90.000,E1 61.051} C_DIS
LIN {X -0.152,Y -548.823,Z 641.138,A 0.000,B 0.000,C 90.000,E1 60.795} C_DIS
LIN {X 0.111,Y -543.883,Z 641.135,A 0.000,B 0.000,C 90.000,E1 60.205} C_DIS
LIN {X 0.097,Y -539.700,Z 641.132,A 0.000,B 0.000,C 90.000,E1 59.793} C_DIS
LIN {X 0.063,Y -534.024,Z 641.129,A 0.000,B 0.000,C 90.000,E1 59.282} C_DIS
LIN {X -0.045,Y -527.816,Z 641.127,A 0.000,B 0.000,C 90.000,E1 58.820} C_DIS
LIN {X 0.257,Y -523.074,Z 641.125,A 0.000,B 0.000,C 90.000,E1 58.456} C_DIS
LIN {X -0.046,Y -516.275,Z 641.123,A 0.000,B 0.000,C 90.000,E1 58.074} C_DIS
LIN {X 0.038,Y -506.360,Z 641.120,A 0.000,B 0.000,C 90.000,E1 57.502} C_DIS
LIN {X -0.023,Y -482.582,Z 641.113,A 0.000,B 0.000,C 90.000,E1 56.294} C_DIS
LIN {X -0.236,Y -460.520,Z 641.106,A 0.000,B 0.000,C 90.000,E1 55.182} C_DIS
LIN {X -0.115,Y -437.675,Z 641.099,A 0.000,B 0.000,C 90.000,E1 53.909} C_DIS
LIN {X -0.137,Y -437.631,Z 641.099,A 0.000,B 0.000,C 90.000,E1 53.909} C_DIS
LIN {X -0.139,Y -431.444,Z 641.082,A 0.000,B 0.000,C 90.000,E1 50.803} C_DIS
LIN {X 0.020,Y -423.267,Z 641.063,A 0.000,B 0.000,C 90.000,E1 47.268} C_DIS
LIN {X 0.271,Y -423.613,Z 641.056,A 0.000,B 0.000,C 90.000,E1 46.053} C_DIS
LIN {X -0.019,Y -423.825,Z 641.050,A 0.000,B 0.000,C 90.000,E1 45.081} C_DIS
LIN {X 0.118,Y -424.247,Z 641.036,A 0.000,B 0.000,C 90.000,E1 42.366} C_DIS
LIN {X -0.121,Y -424.873,Z 641.024,A 0.000,B 0.000,C 90.000,E1 40.378} C_DIS
LIN {X 0.159,Y -426.026,Z 641.009,A 0.000,B 0.000,C 90.000,E1 37.649} C_DIS
LIN {X 0.065,Y -427.203,Z 640.996,A 0.000,B 0.000,C 90.000,E1 35.311} C_DIS
LIN {X 0.120,Y -428.075,Z 640.985,A 0.000,B 0.000,C 90.000,E1 33.293} C_DIS
LIN {X -0.270,Y -428.824,Z 640.976,A 0.000,B 0.000,C 90.000,E1 31.671} C_DIS
LIN {X 0.092,Y -429.554,Z 640.966,A 0.000,B 0.000,C 90.000,E1 29.951} C_DIS
LIN {X -0.113,Y -430.444,Z 640.955,A 0.000,B 0.000,C 90.000,E1 27.975} C_DIS
LIN {X -0.126,Y -431.428,Z 640.944,A 0.000,B 0.000,C 90.000,E1 25.976} C_DIS
LIN {X -0.103,Y -432.785,Z 640.931,A 0.000,B 0.000,C 90.000,E1 23.643} C_DIS
LIN {X -0.047,Y -434.088,Z 640.920,A 0.000,B 0.000,C 90.000,E1 21.642} C_DIS
LIN {X 0.061,Y -434.951,Z 640.913,A 0.000,B 0.000,C 90.000,E1 20.301} C_DIS
LIN {X -0.129,Y -435.939,Z 640.904,A 0.000,B 0.000,C 90.000,E1 18.671} C_DIS
LIN {X 0.120,Y -436.893,Z 640.894,A 0.000,B 0.000,C 90.000,E1 16.985} C_DIS
LIN {X 0.087,Y -438.153,Z 640.883,A 0.000,B 0.000,C 90.000,E1 15.009} C_DIS
LIN {X -0.149,Y -439.654,Z 640.872,A 0.000,B 0.000,C 90.000,E1 13.063} C_DIS
LIN {X -0.051,Y -441.798,Z 640.858,A 0.000,B 0.000,C 90.000,E1 10.423} C_DIS
LIN {X 0.037,Y -444.668,Z 640.842,A 0.000,B 0.000,C 90.000,E1 7.466} C_DIS
LIN {X 0.203,Y -447.065,Z 640.829,A 0.000,B 0.000,C 90.000,E1 5.163} C_DIS
LIN {X -0.046,Y -449.808,Z 640.816,A 0.000,B 0.000,C 90.000,E1 2.922} C_DIS
LIN {X 0.184,Y -452.744,Z 640.804,A 0.000,B 0.000,C 90.000,E1 0.630} C_DIS
LIN {X -0.113,Y -456.855,Z 640.788,A 0.000,B 0.000,C 90.000,E1 357.879} C_DIS
LIN {X -0.070,Y -459.496,Z 640.779,A 0.000,B 0.000,C 90.000,E1 356.274} C_DIS
LIN {X -0.174,Y -462.722,Z 640.769,A 0.000,B 0.000,C 90.000,E1 354.375} C_DIS
LIN {X 0.052,Y -465.529,Z 640.760,A 0.000,B 0.000,C 90.000,E1 352.761} C_DIS
LIN {X 0.204,Y -468.796,Z 640.749,A 0.000,B 0.000,C 90.000,E1 350.849} C_DIS
LIN {X -0.148,Y -471.015,Z 640.742,A 0.000,B 0.000,C 90.000,E1 349.634} C_DIS
LIN {X 0.129,Y -474.766,Z 640.730,A 0.000,B 0.000,C 90.000,E1 347.409} C_DIS
LIN {X -0.152,Y -478.153,Z 640.720,A 0.000,B 0.000,C 90.000,E1 345.574} C_DIS
LIN {X 0.258,Y -481.056,Z 640.711,A 0.000,B 0.000,C 90.000,E1 343.976} C_DIS
LIN {X -0.216,Y -484.619,Z 640.701,A 0.000,B 0.000,C 90.000,E1 342.181} C_DIS
LIN {X 0.135,Y -487.611,Z 640.692,A 0.000,B 0.000,C 90.000,E1 340.604} C_DIS
LIN {X 0.150,Y -491.852,Z 640.680,A 0.000,B 0.000,C 90.000,E1 338.465} C_DIS
LIN {X 0.267,Y -493.566,Z 640.675,A 0.000,B 0.000,C 90.000,E1 337.539} C_DIS
LIN {X -0.006,Y -495.607,Z 640.669,A 0.000,B 0.000,C 90.000,E1 336.357} C_DIS
LIN {X -0.308,Y -497.117,Z 640.664,A 0.000,B 0.000,C 90.000,E1 335.485} C_DIS
LIN {X 0.061,Y -500.439,Z 640.652,A 0.000,B 0.000,C 90.000,E1 333.332} C_DIS
LIN {X -0.154,Y -503.770,Z 640.640,A 0.000,B 0.000,C 90.000,E1 331.257} C_DIS
LIN {X -0.153,Y -508.188,Z 640.627,A 0.000,B 0.000,C 90.000,E1 328.869} C_DIS
LIN {X 0.031,Y -511.223,Z 640.620,A 0.000,B 0.000,C 90.000,E1 327.661} C_DIS
LIN {X 0.277,Y -513.372,Z 640.617,A 0.000,B 0.000,C 90.000,E1 327.041} C_DIS
LIN {X 0.027,Y -515.036,Z 640.615,A 0.000,B 0.000,C 90.000,E1 326.707} C_DIS
LIN {X 0.205,Y -518.031,Z 640.612,A 0.000,B 0.000,C 90.000,E1 326.215} C_DIS
LIN {X 0.139,Y -520.318,Z 640.611,A 0.000,B 0.000,C 90.000,E1 325.928} C_DIS
LIN {X 0.026,Y -524.484,Z 640.608,A 0.000,B 0.000,C 90.000,E1 325.515} C_DIS
LIN {X -0.009,Y -545.577,Z 640.599,A 0.000,B 0.000,C 90.000,E1 323.783} C_DIS
LIN {X 0.015,Y -554.056,Z 640.595,A 0.000,B 0.000,C 90.000,E1 323.084} C_DIS
LIN {X -0.296,Y -563.860,Z 640.590,A 0.000,B 0.000,C 90.000,E1 322.271} C_DIS
LIN {X -0.100,Y -573.291,Z 640.586,A 0.000,B 0.000,C 90.000,E1 321.412} C_DIS
LIN {X -0.157,Y -582.834,Z 640.581,A 0.000,B 0.000,C 90.000,E1 320.561} C_DIS
LIN {X -0.140,Y -592.187,Z 640.576,A 0.000,B 0.000,C 90.000,E1 319.703} C_DIS
LIN {X -0.154,Y -601.065,Z 640.571,A 0.000,B 0.000,C 90.000,E1 318.852} C_DIS
LIN {X 0.138,Y -604.931,Z 640.569,A 0.000,B 0.000,C 90.000,E1 318.447} C_DIS
LIN {X 0.032,Y -613.291,Z 640.564,A 0.000,B 0.000,C 90.000,E1 317.553} C_DIS
LIN {X 0.045,Y -618.767,Z 640.561,A 0.000,B 0.000,C 90.000,E1 316.905} C_DIS
LIN {X -0.176,Y -621.890,Z 640.559,A 0.000,B 0.000,C 90.000,E1 316.539} C_DIS
LIN {X -0.221,Y -628.704,Z 640.554,A 0.000,B 0.000,C 90.000,E1 315.648} C_DIS
LIN {X 0.214,Y -636.017,Z 640.548,A 0.000,B 0.000,C 90.000,E1 314.595} C_DIS
LIN {X 0.258,Y -643.816,Z 640.542,A 0.000,B 0.000,C 90.000,E1 313.461} C_DIS
LIN {X 0.028,Y -649.686,Z 640.537,A 0.000,B 0.000,C 90.000,E1 312.609} C_DIS
LIN {X -0.090,Y -653.663,Z 640.533,A 0.000,B 0.000,C 90.000,E1 312.000} C_DIS
LIN {X -0.209,Y -659.010,Z 640.529,A 0.000,B 0.000,C 90.000,E1 311.148} C_DIS
LIN {X -0.253,Y -662.401,Z 640.525,A 0.000,B 0.000,C 90.000,E1 310.539} C_DIS
LIN {X -0.269,Y -665.568,Z 640.522,A 0.000,B 0.000,C 90.000,E1 309.930} C_DIS
LIN {X -0.251,Y -667.418,Z 640.520,A 0.000,B 0.000,C 90.000,E1 309.564} C_DIS
LIN {X -0.188,Y -670.759,Z 640.516,A 0.000,B 0.000,C 90.000,E1 308.830} C_DIS
LIN {X -0.091,Y -672.827,Z 640.513,A 0.000,B 0.000,C 90.000,E1 308.338} C_DIS
LIN {X 0.027,Y -675.676,Z 640.509,A 0.000,B 0.000,C 90.000,E1 307.604} C_DIS
LIN {X 0.172,Y -678.306,Z 640.505,A 0.000,B 0.000,C 90.000,E1 306.870} C_DIS
LIN {X -0.058,Y -681.506,Z 640.500,A 0.000,B 0.000,C 90.000,E1 305.931} C_DIS
LIN {X -0.090,Y -684.505,Z 640.494,A 0.000,B 0.000,C 90.000,E1 304.978} C_DIS
LIN {X -0.056,Y -688.057,Z 640.488,A 0.000,B 0.000,C 90.000,E1 303.785} C_DIS
LIN {X 0.010,Y -690.678,Z 640.482,A 0.000,B 0.000,C 90.000,E1 302.832} C_DIS
LIN {X -0.246,Y -693.710,Z 640.476,A 0.000,B 0.000,C 90.000,E1 301.671} C_DIS
LIN {X -0.117,Y -696.034,Z 640.471,A 0.000,B 0.000,C 90.000,E1 300.718} C_DIS
LIN {X -0.058,Y -698.717,Z 640.464,A 0.000,B 0.000,C 90.000,E1 299.539} C_DIS
LIN {X -0.222,Y -700.615,Z 640.459,A 0.000,B 0.000,C 90.000,E1 298.615} C_DIS
LIN {X 0.251,Y -702.358,Z 640.454,A 0.000,B 0.000,C 90.000,E1 297.641} C_DIS
LIN {X 0.145,Y -703.524,Z 640.450,A 0.000,B 0.000,C 90.000,E1 296.950} C_DIS
LIN {X 0.369,Y -704.395,Z 640.446,A 0.000,B 0.000,C 90.000,E1 296.232} C_DIS
LIN {X -0.347,Y -704.643,Z 640.442,A 0.000,B 0.000,C 90.000,E1 295.591} C_DIS
LIN {X 0.226,Y -703.636,Z 640.439,A 0.000,B 0.000,C 90.000,E1 295.079} C_DIS
